KUKA KRL program: EPS_2_251806_MH42A_A_20260212042235.src

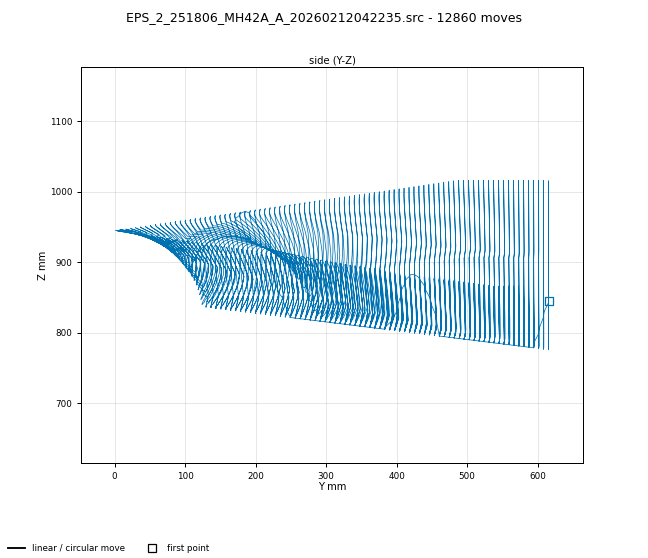
[picture p0: tool path of EPS_2_251806_MH42A_A_20260212042235.src, 12860 of 12862 moves have a stored position in this frame; points joined in program order, loops and branches not executed]
&ACCESS RVP
&REL 4
&COMMENT QRS 19112012
&PARAM EDITMASK = *
DEF PART()
EXT BAS (BAS_COMMAND :IN,REAL :IN )
INT I
BAS (#INITMOV,0 )

;KUKA QRS Post kuka4.cps  Date:22-06-2017 !

File_ID=3014

QRS_PRE_INIT()

;Init var - Until changes are made in qrs_pre_init
Outlet_Square_prg=0
Inlet_1_Square_prg=0
Inlet_2_Square_prg=0
Inlet_3_Square_prg=0
Inlet_4_Square_prg=0
Inlet_5_Square_prg=0

Outlet_1={X 0.000, Y 487.620, Z 915.500, B 0.000, E1 0.000 }
Inlet_1={X 0.000, Y 518.170, Z 495.500, B 0.000, E1 90.000 }
Inlet_2={X 0.000, Y 534.120, Z 275.500, B 0.000, E1 180.000 }
Outlet_1_type=201
Inlet_1_type=201
Inlet_2_type=201
;QRS#1=Sidecore dimensions
;QRS#2=200-8" PVC SDR 35
;QRS#3=200-8" PVC SDR 35
;QRS#4=200-8" PVC SDR 35
;QRS#5=
;QRS#6=
;QRS#7=
;QRS#8=
;QRS#9=12-08 PSX
;QRS#10=12-08 PSX
;QRS#11=12-08 PSX
;QRS#12=
;QRS#13=
;QRS#14=
;QRS#15=
;QRS#16=1220x127x1295 4,25'
;QRS#17=EPS Height
;QRS#18=1016
;QRS#19=*
;QRS#20= UPDATED VERSION 22-06-2017
;QRS#21=*
Outlet_Square=0100
Inlet_1_Square=0100
Inlet_2_Square=0100
Inlet_3_Square=0
Inlet_4_Square=0
Inlet_5_Square=0
Mill_Square=1
Outlet_Square_Prg=204
Inlet_1_Square_prg=204
Inlet_2_Square_prg=204

QRS_INIT()

$ADVANCE=5

; T1
PTP {E1 173.421,E2 173.421}
PTP {X 0,Y 615.492,A -85,B 0,C 180,E1 173.421,E2 173.421,E3 0,E4 0,E5 0,E6 0}
QRS_SPEED_INIT()
LIN {X 0,Y 615.492,Z 844.236,A -85,B 0,C 180,E1 173.421,E2 173.421,E3 0,E4 0,E5 0,E6 0} C_VEL
LIN {X 0,Y 615.497,Z 836.536,A -85,B 0,C 180,E1 172.455,E2 172.455} C_VEL
LIN {X 0,Y 615.498,Z 826.758,A -85,B 0,C 180,E1 171.463,E2 171.463} C_VEL
LIN {X 0,Y 615.497,Z 816.492,A -85,B 0,C 180,E1 170.636,E2 170.636} C_VEL
LIN {X 0,Y 615.425,Z 804.939,A -85,B 0,C 180,E1 169.888,E2 169.888} C_VEL
LIN {X 0,Y 615.422,Z 793.42,A -85,B 0,C 180,E1 169.306,E2 169.306} C_VEL
LIN {X 0,Y 615.465,Z 781.457,A -85,B 0,C 180,E1 168.848,E2 168.848} C_VEL
LIN {X 0,Y 615.493,Z 775.695,A -85,B 0,C 180,E1 168.661,E2 168.661} C_VEL
LIN {X 0,Y 615.444,Z 775.7,A -85,B 0,C 180,E1 166.085,E2 166.085} C_VEL
LIN {X 0,Y 615.403,Z 775.7,A -85,B 0,C 180,E1 163.411,E2 163.411} C_VEL
LIN {X 0,Y 615.452,Z 775.7,A -85,B 0,C 180,E1 160.661,E2 160.661} C_VEL
LIN {X 0,Y 615.44,Z 775.698,A -85,B 0,C 180,E1 157.862,E2 157.862} C_VEL
LIN {X 0,Y 615.435,Z 775.697,A -85,B 0,C 180,E1 155.726,E2 155.726} C_VEL
LIN {X 0,Y 615.428,Z 775.696,A -85,B 0,C 180,E1 153.553,E2 153.553} C_VEL
LIN {X 0,Y 615.422,Z 775.696,A -85,B 0,C 180,E1 151.338,E2 151.338} C_VEL
LIN {X 0,Y 615.421,Z 775.696,A -85,B 0,C 180,E1 149.076,E2 149.076} C_VEL
LIN {X 0,Y 615.455,Z 775.698,A -85,B 0,C 180,E1 146.471,E2 146.471} C_VEL
LIN {X 0,Y 615.47,Z 775.69,A -85,B 0,C 180,E1 143.574,E2 143.574} C_VEL
LIN {X 0,Y 615.434,Z 775.693,A -85,B 0,C 180,E1 140.945,E2 140.945} C_VEL
LIN {X 0,Y 615.446,Z 775.696,A -85,B 0,C 180,E1 138.522,E2 138.522} C_VEL
LIN {X 0,Y 615.495,Z 775.696,A -85,B 0,C 180,E1 135.851,E2 135.851} C_VEL
LIN {X 0,Y 615.457,Z 775.688,A -85,B 0,C 180,E1 133.044,E2 133.044} C_VEL
LIN {X 0,Y 615.447,Z 775.692,A -85,B 0,C 180,E1 130.61,E2 130.61} C_VEL
LIN {X 0,Y 615.476,Z 775.699,A -85,B 0,C 180,E1 128.01,E2 128.01} C_VEL
LIN {X 0,Y 615.492,Z 775.695,A -85,B 0,C 180,E1 125.616,E2 125.616} C_VEL
LIN {X 0,Y 615.487,Z 775.686,A -85,B 0,C 180,E1 123.237,E2 123.237} C_VEL
LIN {X 0,Y 615.481,Z 775.683,A -85,B 0,C 180,E1 120.921,E2 120.921} C_VEL
LIN {X 0,Y 615.463,Z 775.688,A -85,B 0,C 180,E1 118.445,E2 118.445} C_VEL
LIN {X 0,Y 615.492,Z 775.699,A -85,B 0,C 180,E1 115.716,E2 115.716} C_VEL
LIN {X 0,Y 615.492,Z 775.681,A -85,B 0,C 180,E1 112.845,E2 112.845} C_VEL
LIN {X 0,Y 615.467,Z 775.692,A -85,B 0,C 180,E1 110.034,E2 110.034} C_VEL
LIN {X 0,Y 615.484,Z 775.695,A -85,B 0,C 180,E1 107.272,E2 107.272} C_VEL
LIN {X 0,Y 615.492,Z 775.68,A -85,B 0,C 180,E1 104.55,E2 104.55} C_VEL
LIN {X 0,Y 615.474,Z 775.691,A -85,B 0,C 180,E1 101.862,E2 101.862} C_VEL
LIN {X 0,Y 615.485,Z 775.703,A -85,B 0,C 180,E1 101.236,E2 101.236} C_VEL
LIN {X 0,Y 615.474,Z 787.797,A -85,B 0,C 180,E1 100.836,E2 100.836} C_VEL
LIN {X 0,Y 615.486,Z 800.177,A -85,B 0,C 180,E1 100.279,E2 100.279} C_VEL
LIN {X 0,Y 615.484,Z 811.562,A -85,B 0,C 180,E1 99.614,E2 99.614} C_VEL
LIN {X 0,Y 615.498,Z 821.809,A -85,B 0,C 180,E1 98.868,E2 98.868} C_VEL
LIN {X 0,Y 615.498,Z 830.91,A -85,B 0,C 180,E1 98.042,E2 98.042} C_VEL
LIN {X 0,Y 615.497,Z 838.588,A -85,B 0,C 180,E1 97.217,E2 97.217} C_VEL
LIN {X 0,Y 615.497,Z 846.003,A -85,B 0,C 180,E1 96.228,E2 96.228} C_VEL
LIN {X 0,Y 615.497,Z 851.952,A -85,B 0,C 180,E1 95.242,E2 95.242} C_VEL
LIN {X 0,Y 615.493,Z 856.653,A -85,B 0,C 180,E1 94.258,E2 94.258} C_VEL
LIN {X 0,Y 615.494,Z 860.251,A -85,B 0,C 180,E1 93.274,E2 93.274} C_VEL
LIN {X 0,Y 615.496,Z 862.112,A -85,B 0,C 180,E1 92.619,E2 92.619} C_VEL
LIN {X 0,Y 615.497,Z 863.532,A -85,B 0,C 180,E1 91.964,E2 91.964} C_VEL
LIN {X 0,Y 615.496,Z 865.141,A -85,B 0,C 180,E1 90.655,E2 90.655} C_VEL
LIN {X 0,Y 615.495,Z 865.384,A -85,B 0,C 180,E1 90.001,E2 90.001} C_VEL
LIN {X 0,Y 615.495,Z 865.206,A -85,B 0,C 180,E1 89.347,E2 89.347} C_VEL
LIN {X 0,Y 615.497,Z 863.685,A -85,B 0,C 180,E1 88.038,E2 88.038} C_VEL
LIN {X 0,Y 615.498,Z 862.344,A -85,B 0,C 180,E1 87.383,E2 87.383} C_VEL
LIN {X 0,Y 615.496,Z 859.498,A -85,B 0,C 180,E1 86.401,E2 86.401} C_VEL
LIN {X 0,Y 615.499,Z 855.64,A -85,B 0,C 180,E1 85.417,E2 85.417} C_VEL
LIN {X 0,Y 615.498,Z 850.658,A -85,B 0,C 180,E1 84.432,E2 84.432} C_VEL
LIN {X 0,Y 615.489,Z 844.254,A -85,B 0,C 180,E1 83.424,E2 83.424} C_VEL
LIN {X 0,Y 615.497,Z 836.548,A -85,B 0,C 180,E1 82.456,E2 82.456} C_VEL
LIN {X 0,Y 615.498,Z 826.773,A -85,B 0,C 180,E1 81.465,E2 81.465} C_VEL
LIN {X 0,Y 615.498,Z 816.511,A -85,B 0,C 180,E1 80.637,E2 80.637} C_VEL
LIN {X 0,Y 615.486,Z 804.953,A -85,B 0,C 180,E1 79.89,E2 79.89} C_VEL
LIN {X 0,Y 615.473,Z 793.219,A -85,B 0,C 180,E1 79.299,E2 79.299} C_VEL
LIN {X 0,Y 615.472,Z 781.426,A -85,B 0,C 180,E1 78.847,E2 78.847} C_VEL
LIN {X 0,Y 615.483,Z 775.697,A -85,B 0,C 180,E1 78.662,E2 78.662} C_VEL
LIN {X 0,Y 615.482,Z 775.692,A -85,B 0,C 180,E1 76.071,E2 76.071} C_VEL
LIN {X 0,Y 615.486,Z 775.681,A -85,B 0,C 180,E1 73.415,E2 73.415} C_VEL
LIN {X 0,Y 615.474,Z 775.692,A -85,B 0,C 180,E1 70.663,E2 70.663} C_VEL
LIN {X 0,Y 615.478,Z 775.692,A -85,B 0,C 180,E1 67.865,E2 67.865} C_VEL
LIN {X 0,Y 615.487,Z 775.681,A -85,B 0,C 180,E1 65.01,E2 65.01} C_VEL
LIN {X 0,Y 615.484,Z 775.703,A -85,B 0,C 180,E1 62.087,E2 62.087} C_VEL
LIN {X 0,Y 615.486,Z 775.696,A -85,B 0,C 180,E1 59.842,E2 59.842} C_VEL
LIN {X 0,Y 615.475,Z 775.691,A -85,B 0,C 180,E1 57.544,E2 57.544} C_VEL
LIN {X 0,Y 615.474,Z 775.686,A -85,B 0,C 180,E1 55.186,E2 55.186} C_VEL
LIN {X 0,Y 615.49,Z 775.68,A -85,B 0,C 180,E1 52.76,E2 52.76} C_VEL
LIN {X 0,Y 615.489,Z 775.697,A -85,B 0,C 180,E1 49.911,E2 49.911} C_VEL
LIN {X 0,Y 615.494,Z 775.699,A -85,B 0,C 180,E1 47.65,E2 47.65} C_VEL
LIN {X 0,Y 615.47,Z 775.687,A -85,B 0,C 180,E1 44.932,E2 44.932} C_VEL
LIN {X 0,Y 615.484,Z 775.687,A -85,B 0,C 180,E1 42.082,E2 42.082} C_VEL
LIN {X 0,Y 615.487,Z 775.694,A -85,B 0,C 180,E1 39.75,E2 39.75} C_VEL
LIN {X 0,Y 615.465,Z 775.691,A -85,B 0,C 180,E1 36.937,E2 36.937} C_VEL
LIN {X 0,Y 615.463,Z 775.688,A -85,B 0,C 180,E1 34.701,E2 34.701} C_VEL
LIN {X 0,Y 615.475,Z 775.683,A -85,B 0,C 180,E1 32.332,E2 32.332} C_VEL
LIN {X 0,Y 615.486,Z 775.697,A -85,B 0,C 180,E1 29.407,E2 29.407} C_VEL
LIN {X 0,Y 615.484,Z 775.698,A -85,B 0,C 180,E1 27.049,E2 27.049} C_VEL
LIN {X 0,Y 615.461,Z 775.687,A -85,B 0,C 180,E1 24.273,E2 24.273} C_VEL
LIN {X 0,Y 615.486,Z 775.69,A -85,B 0,C 180,E1 21.432,E2 21.432} C_VEL
LIN {X 0,Y 615.463,Z 775.695,A -85,B 0,C 180,E1 18.604,E2 18.604} C_VEL
LIN {X 0,Y 615.462,Z 775.687,A -85,B 0,C 180,E1 15.906,E2 15.906} C_VEL
LIN {X 0,Y 615.492,Z 775.689,A -85,B 0,C 180,E1 13.201,E2 13.201} C_VEL
LIN {X 0,Y 615.47,Z 775.697,A -85,B 0,C 180,E1 10.527,E2 10.527} C_VEL
LIN {X 0,Y 615.476,Z 775.698,A -85,B 0,C 180,E1 8.537,E2 8.537} C_VEL
LIN {X 0,Y 615.447,Z 775.691,A -85,B 0,C 180,E1 5.899,E2 5.899} C_VEL
LIN {X 0,Y 615.479,Z 775.685,A -85,B 0,C 180,E1 3.273,E2 3.273} C_VEL
LIN {X 0,Y 615.491,Z 775.697,A -85,B 0,C 180,E1 0.654,E2 0.654} C_VEL
LIN {X 0,Y 615.453,Z 775.696,A -85,B 0,C 180,E1 -1.963,E2 -1.963} C_VEL
LIN {X 0,Y 615.458,Z 775.697,A -85,B 0,C 180,E1 -3.929,E2 -3.929} C_VEL
LIN {X 0,Y 615.465,Z 775.698,A -85,B 0,C 180,E1 -5.899,E2 -5.899} C_VEL
LIN {X 0,Y 615.438,Z 775.693,A -85,B 0,C 180,E1 -8.537,E2 -8.537} C_VEL
LIN {X 0,Y 615.475,Z 775.688,A -85,B 0,C 180,E1 -11.193,E2 -11.193} C_VEL
LIN {X 0,Y 615.483,Z 775.699,A -85,B 0,C 180,E1 -13.939,E2 -13.939} C_VEL
LIN {X 0,Y 615.432,Z 775.695,A -85,B 0,C 180,E1 -16.588,E2 -16.588} C_VEL
LIN {X 0,Y 615.432,Z 775.695,A -85,B 0,C 180,E1 -18.648,E2 -18.648} C_VEL
LIN {X 0,Y 615.43,Z 775.695,A -85,B 0,C 180,E1 -20.733,E2 -20.733} C_VEL
LIN {X 0,Y 615.428,Z 775.695,A -85,B 0,C 180,E1 -22.847,E2 -22.847} C_VEL
LIN {X 0,Y 615.424,Z 775.695,A -85,B 0,C 180,E1 -24.995,E2 -24.995} C_VEL
LIN {X 0,Y 615.427,Z 775.695,A -85,B 0,C 180,E1 -27.18,E2 -27.18} C_VEL
LIN {X 0,Y 615.47,Z 775.692,A -85,B 0,C 180,E1 -29.796,E2 -29.796} C_VEL
LIN {X 0,Y 615.47,Z 775.7,A -85,B 0,C 180,E1 -32.459,E2 -32.459} C_VEL
LIN {X 0,Y 615.437,Z 775.698,A -85,B 0,C 180,E1 -34.818,E2 -34.818} C_VEL
LIN {X 0,Y 615.417,Z 775.697,A -85,B 0,C 180,E1 -37.247,E2 -37.247} C_VEL
LIN {X 0,Y 615.461,Z 775.695,A -85,B 0,C 180,E1 -40.089,E2 -40.089} C_VEL
LIN {X 0,Y 615.431,Z 775.699,A -85,B 0,C 180,E1 -43.044,E2 -43.044} C_VEL
LIN {X 0,Y 615.433,Z 775.699,A -85,B 0,C 180,E1 -45.074,E2 -45.074} C_VEL
LIN {X 0,Y 615.451,Z 775.7,A -85,B 0,C 180,E1 -46.956,E2 -46.956} C_VEL
LIN {X 0,Y 615.415,Z 775.699,A -85,B 0,C 180,E1 -49.39,E2 -49.39} C_VEL
LIN {X 0,Y 615.408,Z 775.699,A -85,B 0,C 180,E1 -51.928,E2 -51.928} C_VEL
LIN {X 0,Y 615.43,Z 775.818,A -85,B 0,C 180,E1 -54.357,E2 -54.357} C_VEL
LIN {X 0,Y 615.479,Z 789.637,A -85,B 0,C 180,E1 -57.155,E2 -57.155} C_VEL
LIN {X 0,Y 615.478,Z 803.332,A -85,B 0,C 180,E1 -59.841,E2 -59.841} C_VEL
LIN {X 0,Y 615.456,Z 817.027,A -85,B 0,C 180,E1 -62.455,E2 -62.455} C_VEL
LIN {X 0,Y 615.491,Z 830.716,A -85,B 0,C 180,E1 -65.01,E2 -65.01} C_VEL
LIN {X 0,Y 615.47,Z 846.347,A -85,B 0,C 180,E1 -67.865,E2 -67.865} C_VEL
LIN {X 0,Y 615.451,Z 860.013,A -85,B 0,C 180,E1 -70.315,E2 -70.315} C_VEL
LIN {X 0,Y 615.481,Z 873.666,A -85,B 0,C 180,E1 -72.731,E2 -72.731} C_VEL
LIN {X 0,Y 615.489,Z 889.253,A -85,B 0,C 180,E1 -75.452,E2 -75.452} C_VEL
LIN {X 0,Y 615.464,Z 905.807,A -85,B 0,C 180,E1 -78.307,E2 -78.307} C_VEL
LIN {X 0,Y 615.477,Z 921.127,A -85,B 0,C 180,E1 -78.6,E2 -78.6} C_VEL
LIN {X 0,Y 615.49,Z 933.53,A -85,B 0,C 180,E1 -78.961,E2 -78.961} C_VEL
LIN {X 0,Y 615.489,Z 946.05,A -85,B 0,C 180,E1 -79.474,E2 -79.474} C_VEL
LIN {X 0,Y 615.485,Z 958.411,A -85,B 0,C 180,E1 -80.139,E2 -80.139} C_VEL
LIN {X 0,Y 615.498,Z 969.249,A -85,B 0,C 180,E1 -80.886,E2 -80.886} C_VEL
LIN {X 0,Y 615.499,Z 978.016,A -85,B 0,C 180,E1 -81.63,E2 -81.63} C_VEL
LIN {X 0,Y 615.498,Z 987.617,A -85,B 0,C 180,E1 -82.621,E2 -82.621} C_VEL
LIN {X 0,Y 615.491,Z 995.213,A -85,B 0,C 180,E1 -83.609,E2 -83.609} C_VEL
LIN {X 0,Y 615.498,Z 1002.211,A -85,B 0,C 180,E1 -84.76,E2 -84.76} C_VEL
LIN {X 0,Y 615.493,Z 1006.857,A -85,B 0,C 180,E1 -85.745,E2 -85.745} C_VEL
LIN {X 0,Y 615.494,Z 1010.403,A -85,B 0,C 180,E1 -86.728,E2 -86.728} C_VEL
LIN {X 0,Y 615.497,Z 1012.236,A -85,B 0,C 180,E1 -87.383,E2 -87.383} C_VEL
LIN {X 0,Y 615.497,Z 1013.61,A -85,B 0,C 180,E1 -88.038,E2 -88.038} C_VEL
LIN {X 0,Y 615.496,Z 1015.174,A -85,B 0,C 180,E1 -89.347,E2 -89.347} C_VEL
LIN {X 0,Y 615.494,Z 1015.389,A -85,B 0,C 180,E1 -90.001,E2 -90.001} C_VEL
LIN {X 0,Y 615.495,Z 1014.579,A -85,B 0,C 180,E1 -91.31,E2 -91.31} C_VEL
LIN {X 0,Y 615.497,Z 1013.606,A -85,B 0,C 180,E1 -91.964,E2 -91.964} C_VEL
LIN {X 0,Y 615.497,Z 1012.23,A -85,B 0,C 180,E1 -92.619,E2 -92.619} C_VEL
LIN {X 0,Y 615.496,Z 1009.346,A -85,B 0,C 180,E1 -93.602,E2 -93.602} C_VEL
LIN {X 0,Y 615.498,Z 1005.437,A -85,B 0,C 180,E1 -94.586,E2 -94.586} C_VEL
LIN {X 0,Y 615.499,Z 1000.399,A -85,B 0,C 180,E1 -95.571,E2 -95.571} C_VEL
LIN {X 0,Y 615.49,Z 993.913,A -85,B 0,C 180,E1 -96.578,E2 -96.578} C_VEL
LIN {X 0,Y 615.497,Z 986.123,A -85,B 0,C 180,E1 -97.546,E2 -97.546} C_VEL
LIN {X 0,Y 615.498,Z 976.245,A -85,B 0,C 180,E1 -98.538,E2 -98.538} C_VEL
LIN {X 0,Y 615.498,Z 965.851,A -85,B 0,C 180,E1 -99.365,E2 -99.365} C_VEL
LIN {X 0,Y 615.485,Z 955.558,A -85,B 0,C 180,E1 -100.029,E2 -100.029} C_VEL
LIN {X 0,Y 615.486,Z 944.115,A -85,B 0,C 180,E1 -100.617,E2 -100.617} C_VEL
LIN {X 0,Y 615.492,Z 932.321,A -85,B 0,C 180,E1 -101.078,E2 -101.078} C_VEL
LIN {X 0,Y 615.474,Z 919.198,A -85,B 0,C 180,E1 -101.445,E2 -101.445} C_VEL
LIN {X 0,Y 615.464,Z 905.793,A -85,B 0,C 180,E1 -101.695,E2 -101.695} C_VEL
LIN {X 0,Y 615.489,Z 889.239,A -85,B 0,C 180,E1 -104.55,E2 -104.55} C_VEL
LIN {X 0,Y 615.481,Z 873.652,A -85,B 0,C 180,E1 -107.272,E2 -107.272} C_VEL
LIN {X 0,Y 615.451,Z 859.999,A -85,B 0,C 180,E1 -109.687,E2 -109.687} C_VEL
LIN {X 0,Y 615.489,Z 845.179,A -85,B 0,C 180,E1 -112.346,E2 -112.346} C_VEL
LIN {X 0,Y 615.491,Z 830.702,A -85,B 0,C 180,E1 -114.992,E2 -114.992} C_VEL
LIN {X 0,Y 615.456,Z 817.013,A -85,B 0,C 180,E1 -117.548,E2 -117.548} C_VEL
LIN {X 0,Y 615.478,Z 803.318,A -85,B 0,C 180,E1 -120.161,E2 -120.161} C_VEL
LIN {X 0,Y 615.479,Z 789.623,A -85,B 0,C 180,E1 -122.847,E2 -122.847} C_VEL
LIN {X 0,Y 615.427,Z 775.7,A -85,B 0,C 180,E1 -125.671,E2 -125.671} C_VEL
LIN {X 0,Y 615.406,Z 775.7,A -85,B 0,C 180,E1 -128.075,E2 -128.075} C_VEL
LIN {X 0,Y 615.41,Z 775.7,A -85,B 0,C 180,E1 -130.613,E2 -130.613} C_VEL
LIN {X 0,Y 615.47,Z 775.7,A -85,B 0,C 180,E1 -133.247,E2 -133.247} C_VEL
LIN {X 0,Y 615.43,Z 775.699,A -85,B 0,C 180,E1 -136.009,E2 -136.009} C_VEL
LIN {X 0,Y 615.447,Z 775.699,A -85,B 0,C 180,E1 -137.925,E2 -137.925} C_VEL
LIN {X 0,Y 615.421,Z 775.699,A -85,B 0,C 180,E1 -140.245,E2 -140.245} C_VEL
LIN {X 0,Y 615.404,Z 775.699,A -85,B 0,C 180,E1 -142.752,E2 -142.752} C_VEL
LIN {X 0,Y 615.428,Z 775.7,A -85,B 0,C 180,E1 -145.308,E2 -145.308} C_VEL
LIN {X 0,Y 615.442,Z 775.698,A -85,B 0,C 180,E1 -148.312,E2 -148.312} C_VEL
LIN {X 0,Y 615.422,Z 775.699,A -85,B 0,C 180,E1 -150.59,E2 -150.59} C_VEL
LIN {X 0,Y 615.407,Z 775.699,A -85,B 0,C 180,E1 -152.971,E2 -152.971} C_VEL
LIN {X 0,Y 615.408,Z 775.699,A -85,B 0,C 180,E1 -155.005,E2 -155.005} C_VEL
LIN {X 0,Y 615.405,Z 775.699,A -85,B 0,C 180,E1 -157.152,E2 -157.152} C_VEL
LIN {X 0,Y 615.409,Z 775.699,A -85,B 0,C 180,E1 -159.464,E2 -159.464} C_VEL
LIN {X 0,Y 615.447,Z 775.701,A -85,B 0,C 180,E1 -162.042,E2 -162.042} C_VEL
LIN {X 0,Y 615.454,Z 775.698,A -85,B 0,C 180,E1 -164.773,E2 -164.773} C_VEL
LIN {X 0,Y 615.408,Z 775.698,A -85,B 0,C 180,E1 -167.468,E2 -167.468} C_VEL
LIN {X 0,Y 615.475,Z 775.741,A -85,B 0,C 180,E1 -168.765,E2 -168.765} C_VEL
LIN {X 0,Y 615.425,Z 788.344,A -85,B 0,C 180,E1 -169.184,E2 -169.184} C_VEL
LIN {X 0,Y 615.408,Z 800.209,A -85,B 0,C 180,E1 -169.721,E2 -169.721} C_VEL
LIN {X 0,Y 615.463,Z 811.581,A -85,B 0,C 180,E1 -170.386,E2 -170.386} C_VEL
LIN {X 0,Y 615.498,Z 821.823,A -85,B 0,C 180,E1 -171.133,E2 -171.133} C_VEL
LIN {X 0,Y 615.498,Z 830.921,A -85,B 0,C 180,E1 -171.959,E2 -171.959} C_VEL
LIN {X 0,Y 615.497,Z 838.597,A -85,B 0,C 180,E1 -172.784,E2 -172.784} C_VEL
LIN {X 0,Y 615.497,Z 846.011,A -85,B 0,C 180,E1 -173.773,E2 -173.773} C_VEL
LIN {X 0,Y 615.497,Z 851.958,A -85,B 0,C 180,E1 -174.759,E2 -174.759} C_VEL
LIN {X 0,Y 615.493,Z 856.658,A -85,B 0,C 180,E1 -175.744,E2 -175.744} C_VEL
LIN {X 0,Y 615.496,Z 860.254,A -85,B 0,C 180,E1 -176.727,E2 -176.727} C_VEL
LIN {X 0,Y 615.496,Z 862.115,A -85,B 0,C 180,E1 -177.382,E2 -177.382} C_VEL
LIN {X 0,Y 615.497,Z 863.534,A -85,B 0,C 180,E1 -178.037,E2 -178.037} C_VEL
LIN {X 0,Y 615.496,Z 865.142,A -85,B 0,C 180,E1 -179.346,E2 -179.346} C_VEL
LIN {X 0,Y 615.494,Z 865.384,A -85,B 0,C 180,E1 -180,E2 -180} C_VEL
LIN {X 0,Y 615.495,Z 865.206,A -85,B 0,C 180,E1 -180.654,E2 -180.654} C_VEL
LIN {X 0,Y 615.496,Z 863.683,A -85,B 0,C 180,E1 -181.963,E2 -181.963} C_VEL
LIN {X 0,Y 615.498,Z 862.341,A -85,B 0,C 180,E1 -182.618,E2 -182.618} C_VEL
LIN {X 0,Y 615.496,Z 859.494,A -85,B 0,C 180,E1 -183.601,E2 -183.601} C_VEL
LIN {X 0,Y 615.498,Z 855.634,A -85,B 0,C 180,E1 -184.585,E2 -184.585} C_VEL
LIN {X 0,Y 615.498,Z 850.651,A -85,B 0,C 180,E1 -185.57,E2 -185.57} C_VEL
LIN {X 0,Y 615.492,Z 844.236,A -85,B 0,C 180,E1 -186.579,E2 -186.579} C_VEL
LIN {X 0,Y 614.826,Z 841.054,A -85,B 0,C 180,E1 -187.028,E2 -187.028} C_VEL
LIN {X 0,Y 611.988,Z 835.48,A -85,B 0,C 180,E1 -187.745,E2 -187.745} C_VEL
LIN {X 0,Y 609.138,Z 829.207,A -85,B 0,C 180,E1 -188.426,E2 -188.426} C_VEL
LIN {X 0,Y 608.477,Z 824.966,A -85,B 0,C 180,E1 -188.816,E2 -188.816} C_VEL
LIN {X 0,Y 608.476,Z 814.391,A -85,B 0,C 180,E1 -189.641,E2 -189.641} C_VEL
LIN {X 0,Y 608.422,Z 803.602,A -85,B 0,C 180,E1 -190.314,E2 -190.314} C_VEL
LIN {X 0,Y 608.444,Z 791.79,A -85,B 0,C 180,E1 -190.893,E2 -190.893} C_VEL
LIN {X 0,Y 608.523,Z 778.958,A -85,B 0,C 180,E1 -191.365,E2 -191.365} C_VEL
LIN {X 0,Y 608.472,Z 776.695,A -85,B 0,C 180,E1 -191.45,E2 -191.45} C_VEL
LIN {X 0,Y 608.419,Z 776.694,A -85,B 0,C 180,E1 -194.039,E2 -194.039} C_VEL
LIN {X 0,Y 608.375,Z 776.696,A -85,B 0,C 180,E1 -196.498,E2 -196.498} C_VEL
LIN {X 0,Y 608.392,Z 776.695,A -85,B 0,C 180,E1 -198.872,E2 -198.872} C_VEL
LIN {X 0,Y 608.439,Z 776.7,A -85,B 0,C 180,E1 -201.693,E2 -201.693} C_VEL
LIN {X 0,Y 608.404,Z 776.693,A -85,B 0,C 180,E1 -204.573,E2 -204.573} C_VEL
LIN {X 0,Y 608.387,Z 776.695,A -85,B 0,C 180,E1 -206.777,E2 -206.777} C_VEL
LIN {X 0,Y 608.481,Z 776.694,A -85,B 0,C 180,E1 -209.779,E2 -209.779} C_VEL
LIN {X 0,Y 608.431,Z 776.69,A -85,B 0,C 180,E1 -212.517,E2 -212.517} C_VEL
LIN {X 0,Y 608.4,Z 776.693,A -85,B 0,C 180,E1 -214.898,E2 -214.898} C_VEL
LIN {X 0,Y 608.431,Z 776.69,A -85,B 0,C 180,E1 -217.153,E2 -217.153} C_VEL
LIN {X 0,Y 608.421,Z 776.693,A -85,B 0,C 180,E1 -219.444,E2 -219.444} C_VEL
LIN {X 0,Y 608.468,Z 776.69,A -85,B 0,C 180,E1 -222.334,E2 -222.334} C_VEL
LIN {X 0,Y 608.431,Z 776.69,A -85,B 0,C 180,E1 -224.799,E2 -224.799} C_VEL
LIN {X 0,Y 608.424,Z 776.69,A -85,B 0,C 180,E1 -227.037,E2 -227.037} C_VEL
LIN {X 0,Y 608.427,Z 776.694,A -85,B 0,C 180,E1 -229.694,E2 -229.694} C_VEL
LIN {X 0,Y 608.465,Z 776.695,A -85,B 0,C 180,E1 -232.253,E2 -232.253} C_VEL
LIN {X 0,Y 608.435,Z 776.689,A -85,B 0,C 180,E1 -235.097,E2 -235.097} C_VEL
LIN {X 0,Y 608.451,Z 776.692,A -85,B 0,C 180,E1 -237.904,E2 -237.904} C_VEL
LIN {X 0,Y 608.473,Z 776.694,A -85,B 0,C 180,E1 -240.22,E2 -240.22} C_VEL
LIN {X 0,Y 608.442,Z 776.688,A -85,B 0,C 180,E1 -243.225,E2 -243.225} C_VEL
LIN {X 0,Y 608.44,Z 776.691,A -85,B 0,C 180,E1 -245.856,E2 -245.856} C_VEL
LIN {X 0,Y 608.465,Z 776.694,A -85,B 0,C 180,E1 -248.307,E2 -248.307} C_VEL
LIN {X 0,Y 608.477,Z 776.684,A -85,B 0,C 180,E1 -251.283,E2 -251.283} C_VEL
LIN {X 0,Y 608.454,Z 776.688,A -85,B 0,C 180,E1 -253.905,E2 -253.905} C_VEL
LIN {X 0,Y 608.459,Z 776.696,A -85,B 0,C 180,E1 -256.642,E2 -256.642} C_VEL
LIN {X 0,Y 608.472,Z 776.695,A -85,B 0,C 180,E1 -258.654,E2 -258.654} C_VEL
LIN {X 0,Y 608.512,Z 788.579,A -85,B 0,C 180,E1 -259.063,E2 -259.063} C_VEL
LIN {X 0,Y 608.498,Z 800.342,A -85,B 0,C 180,E1 -259.602,E2 -259.602} C_VEL
LIN {X 0,Y 608.494,Z 811.769,A -85,B 0,C 180,E1 -260.274,E2 -260.274} C_VEL
LIN {X 0,Y 608.474,Z 822.067,A -85,B 0,C 180,E1 -261.028,E2 -261.028} C_VEL
LIN {X 0,Y 608.464,Z 831.232,A -85,B 0,C 180,E1 -261.865,E2 -261.865} C_VEL
LIN {X 0,Y 608.462,Z 838.957,A -85,B 0,C 180,E1 -262.699,E2 -262.699} C_VEL
LIN {X 0,Y 608.449,Z 846.429,A -85,B 0,C 180,E1 -263.699,E2 -263.699} C_VEL
LIN {X 0,Y 608.462,Z 852.429,A -85,B 0,C 180,E1 -264.697,E2 -264.697} C_VEL
LIN {X 0,Y 608.439,Z 857.174,A -85,B 0,C 180,E1 -265.693,E2 -265.693} C_VEL
LIN {X 0,Y 608.425,Z 860.809,A -85,B 0,C 180,E1 -266.688,E2 -266.688} C_VEL
LIN {X 0,Y 608.425,Z 862.687,A -85,B 0,C 180,E1 -267.351,E2 -267.351} C_VEL
LIN {X 0,Y 608.442,Z 864.125,A -85,B 0,C 180,E1 -268.013,E2 -268.013} C_VEL
LIN {X 0,Y 608.439,Z 865.751,A -85,B 0,C 180,E1 -269.337,E2 -269.337} C_VEL
LIN {X 0,Y 608.435,Z 865.995,A -85,B 0,C 180,E1 -269.999,E2 -269.999} C_VEL
LIN {X 0,Y 608.438,Z 865.816,A -85,B 0,C 180,E1 -270.661,E2 -270.661} C_VEL
LIN {X 0,Y 608.443,Z 864.278,A -85,B 0,C 180,E1 -271.985,E2 -271.985} C_VEL
LIN {X 0,Y 608.426,Z 862.921,A -85,B 0,C 180,E1 -272.647,E2 -272.647} C_VEL
LIN {X 0,Y 608.449,Z 860.046,A -85,B 0,C 180,E1 -273.641,E2 -273.641} C_VEL
LIN {X 0,Y 608.433,Z 856.148,A -85,B 0,C 180,E1 -274.637,E2 -274.637} C_VEL
LIN {X 0,Y 608.449,Z 851.12,A -85,B 0,C 180,E1 -275.633,E2 -275.633} C_VEL
LIN {X 0,Y 608.438,Z 844.804,A -85,B 0,C 180,E1 -276.632,E2 -276.632} C_VEL
LIN {X 0,Y 608.475,Z 836.888,A -85,B 0,C 180,E1 -277.632,E2 -277.632} C_VEL
LIN {X 0,Y 608.472,Z 827.043,A -85,B 0,C 180,E1 -278.634,E2 -278.634} C_VEL
LIN {X 0,Y 608.48,Z 816.734,A -85,B 0,C 180,E1 -279.472,E2 -279.472} C_VEL
LIN {X 0,Y 608.483,Z 805.124,A -85,B 0,C 180,E1 -280.228,E2 -280.228} C_VEL
LIN {X 0,Y 608.497,Z 793.336,A -85,B 0,C 180,E1 -280.825,E2 -280.825} C_VEL
LIN {X 0,Y 608.522,Z 781.413,A -85,B 0,C 180,E1 -281.285,E2 -281.285} C_VEL
LIN {X 0,Y 608.468,Z 776.696,A -85,B 0,C 180,E1 -281.449,E2 -281.449} C_VEL
LIN {X 0,Y 608.47,Z 776.688,A -85,B 0,C 180,E1 -284.036,E2 -284.036} C_VEL
LIN {X 0,Y 608.473,Z 776.684,A -85,B 0,C 180,E1 -286.782,E2 -286.782} C_VEL
LIN {X 0,Y 608.443,Z 776.696,A -85,B 0,C 180,E1 -289.569,E2 -289.569} C_VEL
LIN {X 0,Y 608.475,Z 776.685,A -85,B 0,C 180,E1 -292.404,E2 -292.404} C_VEL
LIN {X 0,Y 608.448,Z 776.688,A -85,B 0,C 180,E1 -294.57,E2 -294.57} C_VEL
LIN {X 0,Y 608.475,Z 776.685,A -85,B 0,C 180,E1 -297.206,E2 -297.206} C_VEL
LIN {X 0,Y 608.466,Z 776.697,A -85,B 0,C 180,E1 -299.971,E2 -299.971} C_VEL
LIN {X 0,Y 608.451,Z 776.69,A -85,B 0,C 180,E1 -302.52,E2 -302.52} C_VEL
LIN {X 0,Y 608.433,Z 776.689,A -85,B 0,C 180,E1 -305.276,E2 -305.276} C_VEL
LIN {X 0,Y 608.471,Z 776.688,A -85,B 0,C 180,E1 -307.744,E2 -307.744} C_VEL
LIN {X 0,Y 608.448,Z 776.697,A -85,B 0,C 180,E1 -310.328,E2 -310.328} C_VEL
LIN {X 0,Y 608.441,Z 776.689,A -85,B 0,C 180,E1 -312.958,E2 -312.958} C_VEL
LIN {X 0,Y 608.451,Z 776.688,A -85,B 0,C 180,E1 -315.734,E2 -315.734} C_VEL
LIN {X 0,Y 608.455,Z 776.694,A -85,B 0,C 180,E1 -318.656,E2 -318.656} C_VEL
LIN {X 0,Y 608.456,Z 776.686,A -85,B 0,C 180,E1 -321.411,E2 -321.411} C_VEL
LIN {X 0,Y 608.468,Z 776.686,A -85,B 0,C 180,E1 -323.949,E2 -323.949} C_VEL
LIN {X 0,Y 608.467,Z 776.69,A -85,B 0,C 180,E1 -326.329,E2 -326.329} C_VEL
LIN {X 0,Y 608.466,Z 776.696,A -85,B 0,C 180,E1 -328.726,E2 -328.726} C_VEL
LIN {X 0,Y 608.449,Z 776.689,A -85,B 0,C 180,E1 -331.38,E2 -331.38} C_VEL
LIN {X 0,Y 608.437,Z 776.688,A -85,B 0,C 180,E1 -333.964,E2 -333.964} C_VEL
LIN {X 0,Y 608.459,Z 776.686,A -85,B 0,C 180,E1 -336.155,E2 -336.155} C_VEL
LIN {X 0,Y 608.444,Z 776.698,A -85,B 0,C 180,E1 -339.018,E2 -339.018} C_VEL
LIN {X 0,Y 608.427,Z 776.69,A -85,B 0,C 180,E1 -341.827,E2 -341.827} C_VEL
LIN {X 0,Y 608.466,Z 776.688,A -85,B 0,C 180,E1 -344.594,E2 -344.594} C_VEL
LIN {X 0,Y 608.461,Z 776.694,A -85,B 0,C 180,E1 -347.323,E2 -347.323} C_VEL
LIN {X 0,Y 608.455,Z 776.695,A -85,B 0,C 180,E1 -349.35,E2 -349.35} C_VEL
LIN {X 0,Y 608.447,Z 776.688,A -85,B 0,C 180,E1 -352.033,E2 -352.033} C_VEL
LIN {X 0,Y 608.461,Z 776.687,A -85,B 0,C 180,E1 -354.698,E2 -354.698} C_VEL
LIN {X 0,Y 608.483,Z 776.693,A -85,B 0,C 180,E1 -357.352,E2 -357.352} C_VEL
LIN {X 0,Y 608.44,Z 776.691,A -85,B 0,C 180,E1 -360,E2 -360} C_VEL
LIN {X 0,Y 608.445,Z 776.688,A -85,B 0,C 180,E1 -362.648,E2 -362.648} C_VEL
LIN {X 0,Y 608.468,Z 776.69,A -85,B 0,C 180,E1 -365.302,E2 -365.302} C_VEL
LIN {X 0,Y 608.459,Z 776.692,A -85,B 0,C 180,E1 -367.967,E2 -367.967} C_VEL
LIN {X 0,Y 608.42,Z 776.691,A -85,B 0,C 180,E1 -370.651,E2 -370.651} C_VEL
LIN {X 0,Y 608.451,Z 776.69,A -85,B 0,C 180,E1 -373.357,E2 -373.357} C_VEL
LIN {X 0,Y 608.441,Z 776.695,A -85,B 0,C 180,E1 -376.094,E2 -376.094} C_VEL
LIN {X 0,Y 608.421,Z 776.69,A -85,B 0,C 180,E1 -378.871,E2 -378.871} C_VEL
LIN {X 0,Y 608.45,Z 776.692,A -85,B 0,C 180,E1 -381.692,E2 -381.692} C_VEL
LIN {X 0,Y 608.419,Z 776.694,A -85,B 0,C 180,E1 -384.573,E2 -384.573} C_VEL
LIN {X 0,Y 608.406,Z 776.692,A -85,B 0,C 180,E1 -387.198,E2 -387.198} C_VEL
LIN {X 0,Y 608.48,Z 776.69,A -85,B 0,C 180,E1 -389.977,E2 -389.977} C_VEL
LIN {X 0,Y 608.417,Z 776.693,A -85,B 0,C 180,E1 -392.882,E2 -392.882} C_VEL
LIN {X 0,Y 608.395,Z 776.694,A -85,B 0,C 180,E1 -395.281,E2 -395.281} C_VEL
LIN {X 0,Y 608.446,Z 776.695,A -85,B 0,C 180,E1 -398.241,E2 -398.241} C_VEL
LIN {X 0,Y 608.391,Z 776.695,A -85,B 0,C 180,E1 -401.182,E2 -401.182} C_VEL
LIN {X 0,Y 608.412,Z 776.692,A -85,B 0,C 180,E1 -403.306,E2 -403.306} C_VEL
LIN {X 0,Y 608.424,Z 776.693,A -85,B 0,C 180,E1 -406.129,E2 -406.129} C_VEL
LIN {X 0,Y 608.437,Z 776.698,A -85,B 0,C 180,E1 -408.824,E2 -408.824} C_VEL
LIN {X 0,Y 608.389,Z 776.696,A -85,B 0,C 180,E1 -411.408,E2 -411.408} C_VEL
LIN {X 0,Y 608.423,Z 776.698,A -85,B 0,C 180,E1 -413.085,E2 -413.085} C_VEL
LIN {X 0,Y 608.417,Z 776.817,A -85,B 0,C 180,E1 -414.091,E2 -414.091} C_VEL
LIN {X 0,Y 608.646,Z 781.454,A -85,B 0,C 180,E1 -415.068,E2 -415.068} C_VEL
LIN {X 0,Y 608.623,Z 794.35,A -85,B 0,C 180,E1 -417.686,E2 -417.686} C_VEL
LIN {X 0,Y 608.582,Z 807.245,A -85,B 0,C 180,E1 -420.228,E2 -420.228} C_VEL
LIN {X 0,Y 608.565,Z 821.69,A -85,B 0,C 180,E1 -423.004,E2 -423.004} C_VEL
LIN {X 0,Y 608.554,Z 835.972,A -85,B 0,C 180,E1 -425.684,E2 -425.684} C_VEL
LIN {X 0,Y 608.475,Z 850.285,A -85,B 0,C 180,E1 -428.31,E2 -428.31} C_VEL
LIN {X 0,Y 608.515,Z 866.713,A -85,B 0,C 180,E1 -431.273,E2 -431.273} C_VEL
LIN {X 0,Y 608.49,Z 881.587,A -85,B 0,C 180,E1 -433.908,E2 -433.908} C_VEL
LIN {X 0,Y 608.431,Z 897.238,A -85,B 0,C 180,E1 -436.644,E2 -436.644} C_VEL
LIN {X 0,Y 608.427,Z 906.189,A -85,B 0,C 180,E1 -438.191,E2 -438.191} C_VEL
LIN {X 0,Y 608.539,Z 919.413,A -85,B 0,C 180,E1 -438.426,E2 -438.426} C_VEL
LIN {X 0,Y 608.527,Z 932.253,A -85,B 0,C 180,E1 -438.787,E2 -438.787} C_VEL
LIN {X 0,Y 608.508,Z 944.298,A -85,B 0,C 180,E1 -439.261,E2 -439.261} C_VEL
LIN {X 0,Y 608.48,Z 955.778,A -85,B 0,C 180,E1 -439.856,E2 -439.856} C_VEL
LIN {X 0,Y 608.503,Z 967.27,A -85,B 0,C 180,E1 -440.612,E2 -440.612} C_VEL
LIN {X 0,Y 608.472,Z 976.551,A -85,B 0,C 180,E1 -441.366,E2 -441.366} C_VEL
LIN {X 0,Y 608.475,Z 986.489,A -85,B 0,C 180,E1 -442.368,E2 -442.368} C_VEL
LIN {X 0,Y 608.441,Z 994.716,A -85,B 0,C 180,E1 -443.401,E2 -443.401} C_VEL
LIN {X 0,Y 608.45,Z 1000.873,A -85,B 0,C 180,E1 -444.367,E2 -444.367} C_VEL
LIN {X 0,Y 608.432,Z 1005.955,A -85,B 0,C 180,E1 -445.363,E2 -445.363} C_VEL
LIN {X 0,Y 608.449,Z 1009.9,A -85,B 0,C 180,E1 -446.359,E2 -446.359} C_VEL
LIN {X 0,Y 608.425,Z 1012.812,A -85,B 0,C 180,E1 -447.353,E2 -447.353} C_VEL
LIN {X 0,Y 608.442,Z 1014.203,A -85,B 0,C 180,E1 -448.015,E2 -448.015} C_VEL
LIN {X 0,Y 608.438,Z 1015.784,A -85,B 0,C 180,E1 -449.339,E2 -449.339} C_VEL
LIN {X 0,Y 608.434,Z 1016,A -85,B 0,C 180,E1 -450.001,E2 -450.001} C_VEL
LIN {X 0,Y 608.448,Z 1015.182,A -85,B 0,C 180,E1 -451.325,E2 -451.325} C_VEL
LIN {X 0,Y 608.442,Z 1014.199,A -85,B 0,C 180,E1 -451.987,E2 -451.987} C_VEL
LIN {X 0,Y 608.425,Z 1012.806,A -85,B 0,C 180,E1 -452.649,E2 -452.649} C_VEL
LIN {X 0,Y 608.449,Z 1009.892,A -85,B 0,C 180,E1 -453.644,E2 -453.644} C_VEL
LIN {X 0,Y 608.432,Z 1005.945,A -85,B 0,C 180,E1 -454.639,E2 -454.639} C_VEL
LIN {X 0,Y 608.437,Z 999.87,A -85,B 0,C 180,E1 -455.802,E2 -455.802} C_VEL
LIN {X 0,Y 608.462,Z 993.227,A -85,B 0,C 180,E1 -456.8,E2 -456.8} C_VEL
LIN {X 0,Y 608.456,Z 984.979,A -85,B 0,C 180,E1 -457.801,E2 -457.801} C_VEL
LIN {X 0,Y 608.477,Z 974.586,A -85,B 0,C 180,E1 -458.804,E2 -458.804} C_VEL
LIN {X 0,Y 608.493,Z 963.731,A -85,B 0,C 180,E1 -459.642,E2 -459.642} C_VEL
LIN {X 0,Y 608.49,Z 952.753,A -85,B 0,C 180,E1 -460.314,E2 -460.314} C_VEL
LIN {X 0,Y 608.507,Z 940.876,A -85,B 0,C 180,E1 -460.886,E2 -460.886} C_VEL
LIN {X 0,Y 608.553,Z 928.848,A -85,B 0,C 180,E1 -461.323,E2 -461.323} C_VEL
LIN {X 0,Y 608.515,Z 916.457,A -85,B 0,C 180,E1 -461.641,E2 -461.641} C_VEL
LIN {X 0,Y 608.428,Z 906.151,A -85,B 0,C 180,E1 -461.811,E2 -461.811} C_VEL
LIN {X 0,Y 608.469,Z 889.399,A -85,B 0,C 180,E1 -464.722,E2 -464.722} C_VEL
LIN {X 0,Y 608.483,Z 873.748,A -85,B 0,C 180,E1 -467.477,E2 -467.477} C_VEL
LIN {X 0,Y 608.452,Z 860.053,A -85,B 0,C 180,E1 -469.923,E2 -469.923} C_VEL
LIN {X 0,Y 608.55,Z 844.404,A -85,B 0,C 180,E1 -472.761,E2 -472.761} C_VEL
LIN {X 0,Y 608.565,Z 828.349,A -85,B 0,C 180,E1 -475.739,E2 -475.739} C_VEL
LIN {X 0,Y 608.535,Z 815.056,A -85,B 0,C 180,E1 -478.263,E2 -478.263} C_VEL
LIN {X 0,Y 608.613,Z 801.401,A -85,B 0,C 180,E1 -480.915,E2 -480.915} C_VEL
LIN {X 0,Y 608.654,Z 789.623,A -85,B 0,C 180,E1 -483.263,E2 -483.263} C_VEL
LIN {X 0,Y 608.637,Z 778.029,A -85,B 0,C 180,E1 -485.642,E2 -485.642} C_VEL
LIN {X 0,Y 608.39,Z 776.698,A -85,B 0,C 180,E1 -485.976,E2 -485.976} C_VEL
LIN {X 0,Y 608.374,Z 776.696,A -85,B 0,C 180,E1 -488.229,E2 -488.229} C_VEL
LIN {X 0,Y 608.381,Z 776.695,A -85,B 0,C 180,E1 -490.321,E2 -490.321} C_VEL
LIN {X 0,Y 608.377,Z 776.696,A -85,B 0,C 180,E1 -492.325,E2 -492.325} C_VEL
LIN {X 0,Y 608.391,Z 776.694,A -85,B 0,C 180,E1 -494.257,E2 -494.257} C_VEL
LIN {X 0,Y 608.384,Z 776.695,A -85,B 0,C 180,E1 -496.701,E2 -496.701} C_VEL
LIN {X 0,Y 608.379,Z 776.696,A -85,B 0,C 180,E1 -498.817,E2 -498.817} C_VEL
LIN {X 0,Y 608.394,Z 776.7,A -85,B 0,C 180,E1 -501.406,E2 -501.406} C_VEL
LIN {X 0,Y 608.435,Z 776.696,A -85,B 0,C 180,E1 -503.957,E2 -503.957} C_VEL
LIN {X 0,Y 608.414,Z 776.694,A -85,B 0,C 180,E1 -506.326,E2 -506.326} C_VEL
LIN {X 0,Y 608.384,Z 776.695,A -85,B 0,C 180,E1 -508.743,E2 -508.743} C_VEL
LIN {X 0,Y 608.381,Z 776.695,A -85,B 0,C 180,E1 -510.975,E2 -510.975} C_VEL
LIN {X 0,Y 608.379,Z 776.696,A -85,B 0,C 180,E1 -513.222,E2 -513.222} C_VEL
LIN {X 0,Y 608.402,Z 776.694,A -85,B 0,C 180,E1 -515.427,E2 -515.427} C_VEL
LIN {X 0,Y 608.436,Z 776.699,A -85,B 0,C 180,E1 -518.307,E2 -518.307} C_VEL
LIN {X 0,Y 608.393,Z 776.694,A -85,B 0,C 180,E1 -521.128,E2 -521.128} C_VEL
LIN {X 0,Y 608.411,Z 776.695,A -85,B 0,C 180,E1 -523.905,E2 -523.905} C_VEL
LIN {X 0,Y 608.436,Z 776.697,A -85,B 0,C 180,E1 -526.643,E2 -526.643} C_VEL
LIN {X 0,Y 608.471,Z 776.694,A -85,B 0,C 180,E1 -528.655,E2 -528.655} C_VEL
LIN {X 0,Y 608.454,Z 788.367,A -85,B 0,C 180,E1 -529.054,E2 -529.054} C_VEL
LIN {X 0,Y 608.422,Z 800.36,A -85,B 0,C 180,E1 -529.602,E2 -529.602} C_VEL
LIN {X 0,Y 608.463,Z 811.785,A -85,B 0,C 180,E1 -530.275,E2 -530.275} C_VEL
LIN {X 0,Y 608.474,Z 822.082,A -85,B 0,C 180,E1 -531.029,E2 -531.029} C_VEL
LIN {X 0,Y 608.464,Z 831.242,A -85,B 0,C 180,E1 -531.866,E2 -531.866} C_VEL
LIN {X 0,Y 608.462,Z 838.964,A -85,B 0,C 180,E1 -532.701,E2 -532.701} C_VEL
LIN {X 0,Y 608.448,Z 846.435,A -85,B 0,C 180,E1 -533.7,E2 -533.7} C_VEL
LIN {X 0,Y 608.462,Z 852.433,A -85,B 0,C 180,E1 -534.698,E2 -534.698} C_VEL
LIN {X 0,Y 608.439,Z 857.177,A -85,B 0,C 180,E1 -535.694,E2 -535.694} C_VEL
LIN {X 0,Y 608.426,Z 860.811,A -85,B 0,C 180,E1 -536.689,E2 -536.689} C_VEL
LIN {X 0,Y 608.425,Z 862.691,A -85,B 0,C 180,E1 -537.352,E2 -537.352} C_VEL
LIN {X 0,Y 608.442,Z 864.127,A -85,B 0,C 180,E1 -538.014,E2 -538.014} C_VEL
LIN {X 0,Y 608.439,Z 865.752,A -85,B 0,C 180,E1 -539.338,E2 -539.338} C_VEL
LIN {X 0,Y 608.434,Z 865.995,A -85,B 0,C 180,E1 -540,E2 -540} C_VEL
LIN {X 0,Y 608.438,Z 865.815,A -85,B 0,C 180,E1 -540.662,E2 -540.662} C_VEL
LIN {X 0,Y 608.441,Z 864.276,A -85,B 0,C 180,E1 -541.986,E2 -541.986} C_VEL
LIN {X 0,Y 608.426,Z 862.917,A -85,B 0,C 180,E1 -542.648,E2 -542.648} C_VEL
LIN {X 0,Y 608.449,Z 860.04,A -85,B 0,C 180,E1 -543.642,E2 -543.642} C_VEL
LIN {X 0,Y 608.433,Z 856.141,A -85,B 0,C 180,E1 -544.638,E2 -544.638} C_VEL
LIN {X 0,Y 608.449,Z 851.111,A -85,B 0,C 180,E1 -545.634,E2 -545.634} C_VEL
LIN {X 0,Y 608.44,Z 844.794,A -85,B 0,C 180,E1 -546.633,E2 -546.633} C_VEL
LIN {X 0,Y 608.476,Z 836.878,A -85,B 0,C 180,E1 -547.633,E2 -547.633} C_VEL
LIN {X 0,Y 608.472,Z 827.03,A -85,B 0,C 180,E1 -548.636,E2 -548.636} C_VEL
LIN {X 0,Y 608.477,Z 824.966,A -85,B 0,C 180,E1 -548.816,E2 -548.816} C_VEL
LIN {X 0,Y 607.807,Z 820.632,A -85,B 0,C 180,E1 -549.187,E2 -549.187} C_VEL
LIN {X 0,Y 604.947,Z 813.391,A -85,B 0,C 180,E1 -549.766,E2 -549.766} C_VEL
LIN {X 0,Y 602.096,Z 805.768,A -85,B 0,C 180,E1 -550.299,E2 -550.299} C_VEL
LIN {X 0,Y 601.441,Z 800.697,A -85,B 0,C 180,E1 -550.592,E2 -550.592} C_VEL
LIN {X 0,Y 601.501,Z 788.677,A -85,B 0,C 180,E1 -551.153,E2 -551.153} C_VEL
LIN {X 0,Y 601.425,Z 777.578,A -85,B 0,C 180,E1 -551.544,E2 -551.544} C_VEL
LIN {X 0,Y 601.375,Z 777.57,A -85,B 0,C 180,E1 -554.207,E2 -554.207} C_VEL
LIN {X 0,Y 601.361,Z 777.572,A -85,B 0,C 180,E1 -556.988,E2 -556.988} C_VEL
LIN {X 0,Y 601.369,Z 777.577,A -85,B 0,C 180,E1 -559.811,E2 -559.811} C_VEL
LIN {X 0,Y 601.348,Z 777.572,A -85,B 0,C 180,E1 -562.589,E2 -562.589} C_VEL
LIN {X 0,Y 601.363,Z 777.57,A -85,B 0,C 180,E1 -564.88,E2 -564.88} C_VEL
LIN {X 0,Y 601.37,Z 777.573,A -85,B 0,C 180,E1 -567.353,E2 -567.353} C_VEL
LIN {X 0,Y 601.405,Z 777.569,A -85,B 0,C 180,E1 -570.165,E2 -570.165} C_VEL
LIN {X 0,Y 601.392,Z 777.566,A -85,B 0,C 180,E1 -572.71,E2 -572.71} C_VEL
LIN {X 0,Y 601.359,Z 777.571,A -85,B 0,C 180,E1 -575.106,E2 -575.106} C_VEL
LIN {X 0,Y 601.394,Z 777.569,A -85,B 0,C 180,E1 -577.422,E2 -577.422} C_VEL
LIN {X 0,Y 601.4,Z 777.576,A -85,B 0,C 180,E1 -579.996,E2 -579.996} C_VEL
LIN {X 0,Y 601.386,Z 777.568,A -85,B 0,C 180,E1 -582.673,E2 -582.673} C_VEL
LIN {X 0,Y 601.404,Z 777.567,A -85,B 0,C 180,E1 -585.479,E2 -585.479} C_VEL
LIN {X 0,Y 601.423,Z 777.568,A -85,B 0,C 180,E1 -588.407,E2 -588.407} C_VEL
LIN {X 0,Y 601.399,Z 777.566,A -85,B 0,C 180,E1 -590.872,E2 -590.872} C_VEL
LIN {X 0,Y 601.395,Z 777.566,A -85,B 0,C 180,E1 -593.416,E2 -593.416} C_VEL
LIN {X 0,Y 601.419,Z 777.571,A -85,B 0,C 180,E1 -596.067,E2 -596.067} C_VEL
LIN {X 0,Y 601.424,Z 777.568,A -85,B 0,C 180,E1 -598.545,E2 -598.545} C_VEL
LIN {X 0,Y 601.418,Z 777.563,A -85,B 0,C 180,E1 -601.372,E2 -601.372} C_VEL
LIN {X 0,Y 601.398,Z 777.566,A -85,B 0,C 180,E1 -603.635,E2 -603.635} C_VEL
LIN {X 0,Y 601.419,Z 777.57,A -85,B 0,C 180,E1 -606.589,E2 -606.589} C_VEL
LIN {X 0,Y 601.428,Z 777.562,A -85,B 0,C 180,E1 -609.477,E2 -609.477} C_VEL
LIN {X 0,Y 601.393,Z 777.575,A -85,B 0,C 180,E1 -612.311,E2 -612.311} C_VEL
LIN {X 0,Y 601.41,Z 777.574,A -85,B 0,C 180,E1 -614.408,E2 -614.408} C_VEL
LIN {X 0,Y 601.418,Z 777.565,A -85,B 0,C 180,E1 -617.171,E2 -617.171} C_VEL
LIN {X 0,Y 601.421,Z 777.574,A -85,B 0,C 180,E1 -618.541,E2 -618.541} C_VEL
LIN {X 0,Y 601.536,Z 789.758,A -85,B 0,C 180,E1 -618.984,E2 -618.984} C_VEL
LIN {X 0,Y 601.502,Z 800.337,A -85,B 0,C 180,E1 -619.48,E2 -619.48} C_VEL
LIN {X 0,Y 601.46,Z 811.771,A -85,B 0,C 180,E1 -620.159,E2 -620.159} C_VEL
LIN {X 0,Y 601.439,Z 822.069,A -85,B 0,C 180,E1 -620.923,E2 -620.923} C_VEL
LIN {X 0,Y 601.403,Z 831.249,A -85,B 0,C 180,E1 -621.769,E2 -621.769} C_VEL
LIN {X 0,Y 601.412,Z 838.964,A -85,B 0,C 180,E1 -622.613,E2 -622.613} C_VEL
LIN {X 0,Y 601.36,Z 846.338,A -85,B 0,C 180,E1 -623.61,E2 -623.61} C_VEL
LIN {X 0,Y 601.373,Z 852.434,A -85,B 0,C 180,E1 -624.634,E2 -624.634} C_VEL
LIN {X 0,Y 601.353,Z 857.177,A -85,B 0,C 180,E1 -625.642,E2 -625.642} C_VEL
LIN {X 0,Y 601.344,Z 860.811,A -85,B 0,C 180,E1 -626.649,E2 -626.649} C_VEL
LIN {X 0,Y 601.324,Z 862.689,A -85,B 0,C 180,E1 -627.319,E2 -627.319} C_VEL
LIN {X 0,Y 601.341,Z 864.122,A -85,B 0,C 180,E1 -627.99,E2 -627.99} C_VEL
LIN {X 0,Y 601.339,Z 865.752,A -85,B 0,C 180,E1 -629.329,E2 -629.329} C_VEL
LIN {X 0,Y 601.336,Z 865.989,A -85,B 0,C 180,E1 -629.999,E2 -629.999} C_VEL
LIN {X 0,Y 601.339,Z 865.816,A -85,B 0,C 180,E1 -630.668,E2 -630.668} C_VEL
LIN {X 0,Y 601.342,Z 864.277,A -85,B 0,C 180,E1 -632.008,E2 -632.008} C_VEL
LIN {X 0,Y 601.326,Z 862.92,A -85,B 0,C 180,E1 -632.678,E2 -632.678} C_VEL
LIN {X 0,Y 601.368,Z 860.045,A -85,B 0,C 180,E1 -633.684,E2 -633.684} C_VEL
LIN {X 0,Y 601.337,Z 856.148,A -85,B 0,C 180,E1 -634.691,E2 -634.691} C_VEL
LIN {X 0,Y 601.373,Z 851.119,A -85,B 0,C 180,E1 -635.7,E2 -635.7} C_VEL
LIN {X 0,Y 601.38,Z 844.799,A -85,B 0,C 180,E1 -636.71,E2 -636.71} C_VEL
LIN {X 0,Y 601.396,Z 836.878,A -85,B 0,C 180,E1 -637.722,E2 -637.722} C_VEL
LIN {X 0,Y 601.416,Z 827.024,A -85,B 0,C 180,E1 -638.737,E2 -638.737} C_VEL
LIN {X 0,Y 601.446,Z 816.73,A -85,B 0,C 180,E1 -639.584,E2 -639.584} C_VEL
LIN {X 0,Y 601.489,Z 805.12,A -85,B 0,C 180,E1 -640.348,E2 -640.348} C_VEL
LIN {X 0,Y 601.522,Z 794.174,A -85,B 0,C 180,E1 -640.915,E2 -640.915} C_VEL
LIN {X 0,Y 601.546,Z 782.436,A -85,B 0,C 180,E1 -641.383,E2 -641.383} C_VEL
LIN {X 0,Y 601.437,Z 777.572,A -85,B 0,C 180,E1 -641.563,E2 -641.563} C_VEL
LIN {X 0,Y 601.421,Z 777.565,A -85,B 0,C 180,E1 -644.204,E2 -644.204} C_VEL
LIN {X 0,Y 601.429,Z 777.563,A -85,B 0,C 180,E1 -646.984,E2 -646.984} C_VEL
LIN {X 0,Y 601.4,Z 777.575,A -85,B 0,C 180,E1 -649.808,E2 -649.808} C_VEL
LIN {X 0,Y 601.414,Z 777.564,A -85,B 0,C 180,E1 -652.604,E2 -652.604} C_VEL
LIN {X 0,Y 601.398,Z 777.565,A -85,B 0,C 180,E1 -654.877,E2 -654.877} C_VEL
LIN {X 0,Y 601.415,Z 777.574,A -85,B 0,C 180,E1 -657.866,E2 -657.866} C_VEL
LIN {X 0,Y 601.424,Z 777.57,A -85,B 0,C 180,E1 -660.162,E2 -660.162} C_VEL
LIN {X 0,Y 601.414,Z 777.565,A -85,B 0,C 180,E1 -662.714,E2 -662.714} C_VEL
LIN {X 0,Y 601.388,Z 777.567,A -85,B 0,C 180,E1 -665.11,E2 -665.11} C_VEL
LIN {X 0,Y 601.43,Z 777.562,A -85,B 0,C 180,E1 -667.417,E2 -667.417} C_VEL
LIN {X 0,Y 601.405,Z 777.571,A -85,B 0,C 180,E1 -669.993,E2 -669.993} C_VEL
LIN {X 0,Y 601.406,Z 777.569,A -85,B 0,C 180,E1 -672.668,E2 -672.668} C_VEL
LIN {X 0,Y 601.415,Z 777.563,A -85,B 0,C 180,E1 -675.481,E2 -675.481} C_VEL
LIN {X 0,Y 601.418,Z 777.574,A -85,B 0,C 180,E1 -678.405,E2 -678.405} C_VEL
LIN {X 0,Y 601.422,Z 777.567,A -85,B 0,C 180,E1 -680.874,E2 -680.874} C_VEL
LIN {X 0,Y 601.432,Z 777.561,A -85,B 0,C 180,E1 -683.732,E2 -683.732} C_VEL
LIN {X 0,Y 601.424,Z 777.573,A -85,B 0,C 180,E1 -686.686,E2 -686.686} C_VEL
LIN {X 0,Y 601.419,Z 777.568,A -85,B 0,C 180,E1 -689.058,E2 -689.058} C_VEL
LIN {X 0,Y 601.41,Z 777.566,A -85,B 0,C 180,E1 -691.372,E2 -691.372} C_VEL
LIN {X 0,Y 601.392,Z 777.566,A -85,B 0,C 180,E1 -693.636,E2 -693.636} C_VEL
LIN {X 0,Y 601.412,Z 777.569,A -85,B 0,C 180,E1 -696.589,E2 -696.589} C_VEL
LIN {X 0,Y 601.408,Z 777.567,A -85,B 0,C 180,E1 -699.477,E2 -699.477} C_VEL
LIN {X 0,Y 601.386,Z 777.568,A -85,B 0,C 180,E1 -702.311,E2 -702.311} C_VEL
LIN {X 0,Y 601.417,Z 777.574,A -85,B 0,C 180,E1 -705.103,E2 -705.103} C_VEL
LIN {X 0,Y 601.395,Z 777.567,A -85,B 0,C 180,E1 -707.857,E2 -707.857} C_VEL
LIN {X 0,Y 601.408,Z 777.565,A -85,B 0,C 180,E1 -709.904,E2 -709.904} C_VEL
LIN {X 0,Y 601.439,Z 777.561,A -85,B 0,C 180,E1 -712.615,E2 -712.615} C_VEL
LIN {X 0,Y 601.427,Z 777.573,A -85,B 0,C 180,E1 -715.308,E2 -715.308} C_VEL
LIN {X 0,Y 601.391,Z 777.568,A -85,B 0,C 180,E1 -717.991,E2 -717.991} C_VEL
LIN {X 0,Y 601.41,Z 777.567,A -85,B 0,C 180,E1 -720,E2 -720} C_VEL
LIN {X 0,Y 601.413,Z 777.564,A -85,B 0,C 180,E1 -722.679,E2 -722.679} C_VEL
LIN {X 0,Y 601.428,Z 777.568,A -85,B 0,C 180,E1 -725.364,E2 -725.364} C_VEL
LIN {X 0,Y 601.419,Z 777.567,A -85,B 0,C 180,E1 -728.061,E2 -728.061} C_VEL
LIN {X 0,Y 601.378,Z 777.568,A -85,B 0,C 180,E1 -730.777,E2 -730.777} C_VEL
LIN {X 0,Y 601.404,Z 777.57,A -85,B 0,C 180,E1 -733.516,E2 -733.516} C_VEL
LIN {X 0,Y 601.399,Z 777.569,A -85,B 0,C 180,E1 -736.288,E2 -736.288} C_VEL
LIN {X 0,Y 601.392,Z 777.566,A -85,B 0,C 180,E1 -739.1,E2 -739.1} C_VEL
LIN {X 0,Y 601.384,Z 777.578,A -85,B 0,C 180,E1 -741.96,E2 -741.96} C_VEL
LIN {X 0,Y 601.428,Z 777.569,A -85,B 0,C 180,E1 -744.295,E2 -744.295} C_VEL
LIN {X 0,Y 601.368,Z 777.569,A -85,B 0,C 180,E1 -747.115,E2 -747.115} C_VEL
LIN {X 0,Y 601.378,Z 777.568,A -85,B 0,C 180,E1 -749.395,E2 -749.395} C_VEL
LIN {X 0,Y 601.383,Z 777.57,A -85,B 0,C 180,E1 -751.728,E2 -751.728} C_VEL
LIN {X 0,Y 601.4,Z 777.573,A -85,B 0,C 180,E1 -754.12,E2 -754.12} C_VEL
LIN {X 0,Y 601.368,Z 777.577,A -85,B 0,C 180,E1 -756.586,E2 -756.586} C_VEL
LIN {X 0,Y 601.364,Z 777.571,A -85,B 0,C 180,E1 -759.13,E2 -759.13} C_VEL
LIN {X 0,Y 601.389,Z 777.567,A -85,B 0,C 180,E1 -761.768,E2 -761.768} C_VEL
LIN {X 0,Y 601.385,Z 777.578,A -85,B 0,C 180,E1 -764.534,E2 -764.534} C_VEL
LIN {X 0,Y 601.344,Z 777.574,A -85,B 0,C 180,E1 -767.326,E2 -767.326} C_VEL
LIN {X 0,Y 601.372,Z 777.57,A -85,B 0,C 180,E1 -769.432,E2 -769.432} C_VEL
LIN {X 0,Y 601.332,Z 777.575,A -85,B 0,C 180,E1 -771.728,E2 -771.728} C_VEL
LIN {X 0,Y 601.359,Z 777.675,A -85,B 0,C 180,E1 -773.807,E2 -773.807} C_VEL
LIN {X 0,Y 601.882,Z 781.409,A -85,B 0,C 180,E1 -774.608,E2 -774.608} C_VEL
LIN {X 0,Y 601.779,Z 794.15,A -85,B 0,C 180,E1 -777.232,E2 -777.232} C_VEL
LIN {X 0,Y 601.715,Z 807.245,A -85,B 0,C 180,E1 -779.854,E2 -779.854} C_VEL
LIN {X 0,Y 601.659,Z 821.297,A -85,B 0,C 180,E1 -782.593,E2 -782.593} C_VEL
LIN {X 0,Y 601.603,Z 834.634,A -85,B 0,C 180,E1 -785.132,E2 -785.132} C_VEL
LIN {X 0,Y 601.533,Z 848.428,A -85,B 0,C 180,E1 -787.704,E2 -787.704} C_VEL
LIN {X 0,Y 601.487,Z 862.023,A -85,B 0,C 180,E1 -790.195,E2 -790.195} C_VEL
LIN {X 0,Y 601.47,Z 875.718,A -85,B 0,C 180,E1 -792.666,E2 -792.666} C_VEL
LIN {X 0,Y 601.427,Z 891.369,A -85,B 0,C 180,E1 -795.451,E2 -795.451} C_VEL
LIN {X 0,Y 601.398,Z 906.189,A -85,B 0,C 180,E1 -798.051,E2 -798.051} C_VEL
LIN {X 0,Y 601.576,Z 918.498,A -85,B 0,C 180,E1 -798.268,E2 -798.268} C_VEL
LIN {X 0,Y 601.558,Z 931.301,A -85,B 0,C 180,E1 -798.624,E2 -798.624} C_VEL
LIN {X 0,Y 601.538,Z 943.853,A -85,B 0,C 180,E1 -799.115,E2 -799.115} C_VEL
LIN {X 0,Y 601.477,Z 955.779,A -85,B 0,C 180,E1 -799.737,E2 -799.737} C_VEL
LIN {X 0,Y 601.461,Z 967.271,A -85,B 0,C 180,E1 -800.501,E2 -800.501} C_VEL
LIN {X 0,Y 601.436,Z 976.552,A -85,B 0,C 180,E1 -801.264,E2 -801.264} C_VEL
LIN {X 0,Y 601.396,Z 986.489,A -85,B 0,C 180,E1 -802.278,E2 -802.278} C_VEL
LIN {X 0,Y 601.38,Z 994.48,A -85,B 0,C 180,E1 -803.29,E2 -803.29} C_VEL
LIN {X 0,Y 601.371,Z 1000.873,A -85,B 0,C 180,E1 -804.3,E2 -804.3} C_VEL
LIN {X 0,Y 601.336,Z 1005.955,A -85,B 0,C 180,E1 -805.309,E2 -805.309} C_VEL
LIN {X 0,Y 601.367,Z 1009.9,A -85,B 0,C 180,E1 -806.316,E2 -806.316} C_VEL
LIN {X 0,Y 601.325,Z 1012.812,A -85,B 0,C 180,E1 -807.322,E2 -807.322} C_VEL
LIN {X 0,Y 601.341,Z 1014.204,A -85,B 0,C 180,E1 -807.992,E2 -807.992} C_VEL
LIN {X 0,Y 601.339,Z 1015.784,A -85,B 0,C 180,E1 -809.332,E2 -809.332} C_VEL
LIN {X 0,Y 601.335,Z 1016,A -85,B 0,C 180,E1 -810.001,E2 -810.001} C_VEL
LIN {X 0,Y 601.347,Z 1015.183,A -85,B 0,C 180,E1 -811.341,E2 -811.341} C_VEL
LIN {X 0,Y 601.341,Z 1014.2,A -85,B 0,C 180,E1 -812.01,E2 -812.01} C_VEL
LIN {X 0,Y 601.325,Z 1012.806,A -85,B 0,C 180,E1 -812.681,E2 -812.681} C_VEL
LIN {X 0,Y 601.367,Z 1009.892,A -85,B 0,C 180,E1 -813.686,E2 -813.686} C_VEL
LIN {X 0,Y 601.336,Z 1005.945,A -85,B 0,C 180,E1 -814.694,E2 -814.694} C_VEL
LIN {X 0,Y 601.372,Z 999.87,A -85,B 0,C 180,E1 -815.87,E2 -815.87} C_VEL
LIN {X 0,Y 601.382,Z 993.227,A -85,B 0,C 180,E1 -816.881,E2 -816.881} C_VEL
LIN {X 0,Y 601.401,Z 984.98,A -85,B 0,C 180,E1 -817.893,E2 -817.893} C_VEL
LIN {X 0,Y 601.435,Z 974.586,A -85,B 0,C 180,E1 -818.908,E2 -818.908} C_VEL
LIN {X 0,Y 601.479,Z 963.732,A -85,B 0,C 180,E1 -819.755,E2 -819.755} C_VEL
LIN {X 0,Y 601.51,Z 952.754,A -85,B 0,C 180,E1 -820.435,E2 -820.435} C_VEL
LIN {X 0,Y 601.531,Z 940.887,A -85,B 0,C 180,E1 -821.013,E2 -821.013} C_VEL
LIN {X 0,Y 601.586,Z 928.848,A -85,B 0,C 180,E1 -821.456,E2 -821.456} C_VEL
LIN {X 0,Y 601.577,Z 916.457,A -85,B 0,C 180,E1 -821.777,E2 -821.777} C_VEL
LIN {X 0,Y 601.399,Z 906.151,A -85,B 0,C 180,E1 -821.951,E2 -821.951} C_VEL
LIN {X 0,Y 601.417,Z 889.399,A -85,B 0,C 180,E1 -824.898,E2 -824.898} C_VEL
LIN {X 0,Y 601.48,Z 873.748,A -85,B 0,C 180,E1 -827.687,E2 -827.687} C_VEL
LIN {X 0,Y 601.456,Z 860.053,A -85,B 0,C 180,E1 -830.165,E2 -830.165} C_VEL
LIN {X 0,Y 601.579,Z 844.402,A -85,B 0,C 180,E1 -833.04,E2 -833.04} C_VEL
LIN {X 0,Y 601.634,Z 829.122,A -85,B 0,C 180,E1 -835.91,E2 -835.91} C_VEL
LIN {X 0,Y 601.678,Z 815.056,A -85,B 0,C 180,E1 -838.615,E2 -838.615} C_VEL
LIN {X 0,Y 601.751,Z 801.86,A -85,B 0,C 180,E1 -841.215,E2 -841.215} C_VEL
LIN {X 0,Y 601.839,Z 789.874,A -85,B 0,C 180,E1 -843.638,E2 -843.638} C_VEL
LIN {X 0,Y 601.805,Z 779.841,A -85,B 0,C 180,E1 -845.727,E2 -845.727} C_VEL
LIN {X 0,Y 601.349,Z 777.578,A -85,B 0,C 180,E1 -846.253,E2 -846.253} C_VEL
LIN {X 0,Y 601.354,Z 777.572,A -85,B 0,C 180,E1 -848.461,E2 -848.461} C_VEL
LIN {X 0,Y 601.36,Z 777.574,A -85,B 0,C 180,E1 -850.88,E2 -850.88} C_VEL
LIN {X 0,Y 601.405,Z 777.573,A -85,B 0,C 180,E1 -853.589,E2 -853.589} C_VEL
LIN {X 0,Y 601.338,Z 777.573,A -85,B 0,C 180,E1 -856.437,E2 -856.437} C_VEL
LIN {X 0,Y 601.346,Z 777.575,A -85,B 0,C 180,E1 -859.12,E2 -859.12} C_VEL
LIN {X 0,Y 601.37,Z 777.58,A -85,B 0,C 180,E1 -861.728,E2 -861.728} C_VEL
LIN {X 0,Y 601.364,Z 777.573,A -85,B 0,C 180,E1 -864.244,E2 -864.244} C_VEL
LIN {X 0,Y 601.361,Z 777.57,A -85,B 0,C 180,E1 -866.682,E2 -866.682} C_VEL
LIN {X 0,Y 601.359,Z 777.57,A -85,B 0,C 180,E1 -869.054,E2 -869.054} C_VEL
LIN {X 0,Y 601.353,Z 777.573,A -85,B 0,C 180,E1 -871.369,E2 -871.369} C_VEL
LIN {X 0,Y 601.394,Z 777.572,A -85,B 0,C 180,E1 -874.381,E2 -874.381} C_VEL
LIN {X 0,Y 601.362,Z 777.574,A -85,B 0,C 180,E1 -876.587,E2 -876.587} C_VEL
LIN {X 0,Y 601.365,Z 777.57,A -85,B 0,C 180,E1 -879.476,E2 -879.476} C_VEL
LIN {X 0,Y 601.36,Z 777.581,A -85,B 0,C 180,E1 -882.311,E2 -882.311} C_VEL
LIN {X 0,Y 601.367,Z 777.571,A -85,B 0,C 180,E1 -885.101,E2 -885.101} C_VEL
LIN {X 0,Y 601.37,Z 777.57,A -85,B 0,C 180,E1 -887.857,E2 -887.857} C_VEL
LIN {X 0,Y 601.433,Z 777.573,A -85,B 0,C 180,E1 -888.542,E2 -888.542} C_VEL
LIN {X 0,Y 601.476,Z 790.483,A -85,B 0,C 180,E1 -889.014,E2 -889.014} C_VEL
LIN {X 0,Y 601.416,Z 801.927,A -85,B 0,C 180,E1 -889.564,E2 -889.564} C_VEL
LIN {X 0,Y 601.434,Z 813.066,A -85,B 0,C 180,E1 -890.245,E2 -890.245} C_VEL
LIN {X 0,Y 601.448,Z 823.116,A -85,B 0,C 180,E1 -891.008,E2 -891.008} C_VEL
LIN {X 0,Y 601.407,Z 832.957,A -85,B 0,C 180,E1 -891.939,E2 -891.939} C_VEL
LIN {X 0,Y 601.389,Z 840.327,A -85,B 0,C 180,E1 -892.783,E2 -892.783} C_VEL
LIN {X 0,Y 601.374,Z 847.501,A -85,B 0,C 180,E1 -893.787,E2 -893.787} C_VEL
LIN {X 0,Y 601.372,Z 852.433,A -85,B 0,C 180,E1 -894.635,E2 -894.635} C_VEL
LIN {X 0,Y 601.353,Z 857.174,A -85,B 0,C 180,E1 -895.643,E2 -895.643} C_VEL
LIN {X 0,Y 601.346,Z 860.809,A -85,B 0,C 180,E1 -896.65,E2 -896.65} C_VEL
LIN {X 0,Y 601.324,Z 862.694,A -85,B 0,C 180,E1 -897.32,E2 -897.32} C_VEL
LIN {X 0,Y 601.341,Z 864.128,A -85,B 0,C 180,E1 -897.991,E2 -897.991} C_VEL
LIN {X 0,Y 601.339,Z 865.753,A -85,B 0,C 180,E1 -899.33,E2 -899.33} C_VEL
LIN {X 0,Y 601.335,Z 865.996,A -85,B 0,C 180,E1 -900,E2 -900} C_VEL
LIN {X 0,Y 601.339,Z 865.815,A -85,B 0,C 180,E1 -900.67,E2 -900.67} C_VEL
LIN {X 0,Y 601.34,Z 864.276,A -85,B 0,C 180,E1 -902.009,E2 -902.009} C_VEL
LIN {X 0,Y 601.326,Z 862.909,A -85,B 0,C 180,E1 -902.68,E2 -902.68} C_VEL
LIN {X 0,Y 601.368,Z 860.033,A -85,B 0,C 180,E1 -903.685,E2 -903.685} C_VEL
LIN {X 0,Y 601.337,Z 856.134,A -85,B 0,C 180,E1 -904.693,E2 -904.693} C_VEL
LIN {X 0,Y 601.373,Z 851.105,A -85,B 0,C 180,E1 -905.701,E2 -905.701} C_VEL
LIN {X 0,Y 601.382,Z 844.79,A -85,B 0,C 180,E1 -906.711,E2 -906.711} C_VEL
LIN {X 0,Y 601.396,Z 836.873,A -85,B 0,C 180,E1 -907.723,E2 -907.723} C_VEL
LIN {X 0,Y 601.417,Z 827.013,A -85,B 0,C 180,E1 -908.738,E2 -908.738} C_VEL
LIN {X 0,Y 601.466,Z 816.708,A -85,B 0,C 180,E1 -909.585,E2 -909.585} C_VEL
LIN {X 0,Y 601.426,Z 805.095,A -85,B 0,C 180,E1 -910.35,E2 -910.35} C_VEL
LIN {X 0,Y 601.441,Z 800.697,A -85,B 0,C 180,E1 -910.592,E2 -910.592} C_VEL
LIN {X 0,Y 600.786,Z 797.296,A -85,B 0,C 180,E1 -910.782,E2 -910.782} C_VEL
LIN {X 0,Y 598.002,Z 791.997,A -85,B 0,C 180,E1 -911.084,E2 -911.084} C_VEL
LIN {X 0,Y 595.217,Z 786.547,A -85,B 0,C 180,E1 -911.357,E2 -911.357} C_VEL
LIN {X 0,Y 594.554,Z 782.914,A -85,B 0,C 180,E1 -911.501,E2 -911.501} C_VEL
LIN {X 0,Y 594.385,Z 778.449,A -85,B 0,C 180,E1 -911.661,E2 -911.661} C_VEL
LIN {X 0,Y 594.337,Z 778.446,A -85,B 0,C 180,E1 -914.378,E2 -914.378} C_VEL
LIN {X 0,Y 594.314,Z 778.452,A -85,B 0,C 180,E1 -917.196,E2 -917.196} C_VEL
LIN {X 0,Y 594.331,Z 778.449,A -85,B 0,C 180,E1 -920.055,E2 -920.055} C_VEL
LIN {X 0,Y 594.322,Z 778.448,A -85,B 0,C 180,E1 -922.969,E2 -922.969} C_VEL
LIN {X 0,Y 594.326,Z 778.449,A -85,B 0,C 180,E1 -925.195,E2 -925.195} C_VEL
LIN {X 0,Y 594.328,Z 778.452,A -85,B 0,C 180,E1 -927.515,E2 -927.515} C_VEL
LIN {X 0,Y 594.369,Z 778.444,A -85,B 0,C 180,E1 -930.324,E2 -930.324} C_VEL
LIN {X 0,Y 594.34,Z 778.444,A -85,B 0,C 180,E1 -932.953,E2 -932.953} C_VEL
LIN {X 0,Y 594.314,Z 778.451,A -85,B 0,C 180,E1 -935.412,E2 -935.412} C_VEL
LIN {X 0,Y 594.372,Z 778.452,A -85,B 0,C 180,E1 -937.942,E2 -937.942} C_VEL
LIN {X 0,Y 594.359,Z 778.443,A -85,B 0,C 180,E1 -940.819,E2 -940.819} C_VEL
LIN {X 0,Y 594.348,Z 778.445,A -85,B 0,C 180,E1 -943.302,E2 -943.302} C_VEL
LIN {X 0,Y 594.366,Z 778.451,A -85,B 0,C 180,E1 -946.161,E2 -946.161} C_VEL
LIN {X 0,Y 594.371,Z 778.441,A -85,B 0,C 180,E1 -949.179,E2 -949.179} C_VEL
LIN {X 0,Y 594.38,Z 778.449,A -85,B 0,C 180,E1 -952.058,E2 -952.058} C_VEL
LIN {X 0,Y 594.353,Z 778.446,A -85,B 0,C 180,E1 -954.677,E2 -954.677} C_VEL
LIN {X 0,Y 594.379,Z 778.44,A -85,B 0,C 180,E1 -957.089,E2 -957.089} C_VEL
LIN {X 0,Y 594.373,Z 778.442,A -85,B 0,C 180,E1 -959.675,E2 -959.675} C_VEL
LIN {X 0,Y 594.382,Z 778.446,A -85,B 0,C 180,E1 -962.539,E2 -962.539} C_VEL
LIN {X 0,Y 594.379,Z 778.443,A -85,B 0,C 180,E1 -964.806,E2 -964.806} C_VEL
LIN {X 0,Y 594.371,Z 778.441,A -85,B 0,C 180,E1 -967.264,E2 -967.264} C_VEL
LIN {X 0,Y 594.372,Z 778.444,A -85,B 0,C 180,E1 -969.945,E2 -969.945} C_VEL
LIN {X 0,Y 594.386,Z 778.445,A -85,B 0,C 180,E1 -972.806,E2 -972.806} C_VEL
LIN {X 0,Y 594.383,Z 778.441,A -85,B 0,C 180,E1 -975.83,E2 -975.83} C_VEL
LIN {X 0,Y 594.369,Z 778.45,A -85,B 0,C 180,E1 -978.424,E2 -978.424} C_VEL
LIN {X 0,Y 594.595,Z 782.611,A -85,B 0,C 180,E1 -978.58,E2 -978.58} C_VEL
LIN {X 0,Y 594.568,Z 793.871,A -85,B 0,C 180,E1 -979.033,E2 -979.033} C_VEL
LIN {X 0,Y 594.471,Z 806.422,A -85,B 0,C 180,E1 -979.698,E2 -979.698} C_VEL
LIN {X 0,Y 594.415,Z 817.784,A -85,B 0,C 180,E1 -980.471,E2 -980.471} C_VEL
LIN {X 0,Y 594.378,Z 827.84,A -85,B 0,C 180,E1 -981.328,E2 -981.328} C_VEL
LIN {X 0,Y 594.348,Z 837.552,A -85,B 0,C 180,E1 -982.354,E2 -982.354} C_VEL
LIN {X 0,Y 594.301,Z 845.423,A -85,B 0,C 180,E1 -983.393,E2 -983.393} C_VEL
LIN {X 0,Y 594.289,Z 852.439,A -85,B 0,C 180,E1 -984.57,E2 -984.57} C_VEL
LIN {X 0,Y 594.27,Z 857.181,A -85,B 0,C 180,E1 -985.59,E2 -985.59} C_VEL
LIN {X 0,Y 594.267,Z 860.814,A -85,B 0,C 180,E1 -986.609,E2 -986.609} C_VEL
LIN {X 0,Y 594.225,Z 862.69,A -85,B 0,C 180,E1 -987.287,E2 -987.287} C_VEL
LIN {X 0,Y 594.24,Z 864.114,A -85,B 0,C 180,E1 -987.966,E2 -987.966} C_VEL
LIN {X 0,Y 594.247,Z 865.131,A -85,B 0,C 180,E1 -988.643,E2 -988.643} C_VEL
LIN {X 0,Y 594.24,Z 865.752,A -85,B 0,C 180,E1 -989.321,E2 -989.321} C_VEL
LIN {X 0,Y 594.239,Z 865.816,A -85,B 0,C 180,E1 -990.676,E2 -990.676} C_VEL
LIN {X 0,Y 594.24,Z 864.277,A -85,B 0,C 180,E1 -992.032,E2 -992.032} C_VEL
LIN {X 0,Y 594.226,Z 862.919,A -85,B 0,C 180,E1 -992.71,E2 -992.71} C_VEL
LIN {X 0,Y 594.289,Z 860.044,A -85,B 0,C 180,E1 -993.728,E2 -993.728} C_VEL
LIN {X 0,Y 594.242,Z 856.147,A -85,B 0,C 180,E1 -994.748,E2 -994.748} C_VEL
LIN {X 0,Y 594.299,Z 851.118,A -85,B 0,C 180,E1 -995.768,E2 -995.768} C_VEL
LIN {X 0,Y 594.315,Z 844.794,A -85,B 0,C 180,E1 -996.79,E2 -996.79} C_VEL
LIN {X 0,Y 594.346,Z 836.869,A -85,B 0,C 180,E1 -997.814,E2 -997.814} C_VEL
LIN {X 0,Y 594.366,Z 828.787,A -85,B 0,C 180,E1 -998.67,E2 -998.67} C_VEL
LIN {X 0,Y 594.419,Z 820.034,A -85,B 0,C 180,E1 -999.441,E2 -999.441} C_VEL
LIN {X 0,Y 594.445,Z 810.586,A -85,B 0,C 180,E1 -1000.128,E2 -1000.128} C_VEL
LIN {X 0,Y 594.541,Z 800.445,A -85,B 0,C 180,E1 -1000.728,E2 -1000.728} C_VEL
LIN {X 0,Y 594.556,Z 788.497,A -85,B 0,C 180,E1 -1001.291,E2 -1001.291} C_VEL
LIN {X 0,Y 594.392,Z 778.448,A -85,B 0,C 180,E1 -1001.659,E2 -1001.659} C_VEL
LIN {X 0,Y 594.39,Z 778.439,A -85,B 0,C 180,E1 -1004.376,E2 -1004.376} C_VEL
LIN {X 0,Y 594.387,Z 778.442,A -85,B 0,C 180,E1 -1007.192,E2 -1007.192} C_VEL
LIN {X 0,Y 594.372,Z 778.446,A -85,B 0,C 180,E1 -1010.052,E2 -1010.052} C_VEL
LIN {X 0,Y 594.363,Z 778.442,A -85,B 0,C 180,E1 -1012.966,E2 -1012.966} C_VEL
LIN {X 0,Y 594.372,Z 778.442,A -85,B 0,C 180,E1 -1015.191,E2 -1015.191} C_VEL
LIN {X 0,Y 594.382,Z 778.444,A -85,B 0,C 180,E1 -1017.525,E2 -1017.525} C_VEL
LIN {X 0,Y 594.383,Z 778.444,A -85,B 0,C 180,E1 -1020.327,E2 -1020.327} C_VEL
LIN {X 0,Y 594.372,Z 778.441,A -85,B 0,C 180,E1 -1022.949,E2 -1022.949} C_VEL
LIN {X 0,Y 594.348,Z 778.445,A -85,B 0,C 180,E1 -1025.407,E2 -1025.407} C_VEL
LIN {X 0,Y 594.384,Z 778.446,A -85,B 0,C 180,E1 -1027.939,E2 -1027.939} C_VEL
LIN {X 0,Y 594.374,Z 778.443,A -85,B 0,C 180,E1 -1030.821,E2 -1030.821} C_VEL
LIN {X 0,Y 594.373,Z 778.444,A -85,B 0,C 180,E1 -1033.84,E2 -1033.84} C_VEL
LIN {X 0,Y 594.369,Z 778.446,A -85,B 0,C 180,E1 -1036.7,E2 -1036.7} C_VEL
LIN {X 0,Y 594.378,Z 778.44,A -85,B 0,C 180,E1 -1039.433,E2 -1039.433} C_VEL
LIN {X 0,Y 594.38,Z 778.448,A -85,B 0,C 180,E1 -1042.39,E2 -1042.39} C_VEL
LIN {X 0,Y 594.37,Z 778.451,A -85,B 0,C 180,E1 -1044.671,E2 -1044.671} C_VEL
LIN {X 0,Y 594.366,Z 778.445,A -85,B 0,C 180,E1 -1047.087,E2 -1047.087} C_VEL
LIN {X 0,Y 594.387,Z 778.438,A -85,B 0,C 180,E1 -1049.668,E2 -1049.668} C_VEL
LIN {X 0,Y 594.376,Z 778.447,A -85,B 0,C 180,E1 -1052.539,E2 -1052.539} C_VEL
LIN {X 0,Y 594.369,Z 778.451,A -85,B 0,C 180,E1 -1054.806,E2 -1054.806} C_VEL
LIN {X 0,Y 594.35,Z 778.448,A -85,B 0,C 180,E1 -1057.263,E2 -1057.263} C_VEL
LIN {X 0,Y 594.359,Z 778.442,A -85,B 0,C 180,E1 -1059.946,E2 -1059.946} C_VEL
LIN {X 0,Y 594.375,Z 778.447,A -85,B 0,C 180,E1 -1062.806,E2 -1062.806} C_VEL
LIN {X 0,Y 594.37,Z 778.442,A -85,B 0,C 180,E1 -1065.826,E2 -1065.826} C_VEL
LIN {X 0,Y 594.435,Z 778.438,A -85,B 0,C 180,E1 -1068.894,E2 -1068.894} C_VEL
LIN {X 0,Y 594.394,Z 778.44,A -85,B 0,C 180,E1 -1071.843,E2 -1071.843} C_VEL
LIN {X 0,Y 594.381,Z 778.44,A -85,B 0,C 180,E1 -1074.572,E2 -1074.572} C_VEL
LIN {X 0,Y 594.409,Z 778.445,A -85,B 0,C 180,E1 -1077.289,E2 -1077.289} C_VEL
LIN {X 0,Y 594.38,Z 778.442,A -85,B 0,C 180,E1 -1080,E2 -1080} C_VEL
LIN {X 0,Y 594.381,Z 778.44,A -85,B 0,C 180,E1 -1082.711,E2 -1082.711} C_VEL
LIN {X 0,Y 594.388,Z 778.447,A -85,B 0,C 180,E1 -1085.428,E2 -1085.428} C_VEL
LIN {X 0,Y 594.391,Z 778.441,A -85,B 0,C 180,E1 -1088.157,E2 -1088.157} C_VEL
LIN {X 0,Y 594.358,Z 778.443,A -85,B 0,C 180,E1 -1091.068,E2 -1091.068} C_VEL
LIN {X 0,Y 594.366,Z 778.45,A -85,B 0,C 180,E1 -1093.679,E2 -1093.679} C_VEL
LIN {X 0,Y 594.327,Z 778.447,A -85,B 0,C 180,E1 -1096.704,E2 -1096.704} C_VEL
LIN {X 0,Y 594.345,Z 778.446,A -85,B 0,C 180,E1 -1099.335,E2 -1099.335} C_VEL
LIN {X 0,Y 594.339,Z 778.448,A -85,B 0,C 180,E1 -1101.504,E2 -1101.504} C_VEL
LIN {X 0,Y 594.372,Z 778.445,A -85,B 0,C 180,E1 -1104.447,E2 -1104.447} C_VEL
LIN {X 0,Y 594.334,Z 778.447,A -85,B 0,C 180,E1 -1106.702,E2 -1106.702} C_VEL
LIN {X 0,Y 594.355,Z 778.443,A -85,B 0,C 180,E1 -1109,E2 -1109} C_VEL
LIN {X 0,Y 594.356,Z 778.444,A -85,B 0,C 180,E1 -1111.643,E2 -1111.643} C_VEL
LIN {X 0,Y 594.345,Z 778.451,A -85,B 0,C 180,E1 -1114.582,E2 -1114.582} C_VEL
LIN {X 0,Y 594.339,Z 778.445,A -85,B 0,C 180,E1 -1117.605,E2 -1117.605} C_VEL
LIN {X 0,Y 594.346,Z 778.454,A -85,B 0,C 180,E1 -1120.569,E2 -1120.569} C_VEL
LIN {X 0,Y 594.334,Z 778.446,A -85,B 0,C 180,E1 -1123.303,E2 -1123.303} C_VEL
LIN {X 0,Y 594.322,Z 778.451,A -85,B 0,C 180,E1 -1126.165,E2 -1126.165} C_VEL
LIN {X 0,Y 594.347,Z 778.448,A -85,B 0,C 180,E1 -1129.182,E2 -1129.182} C_VEL
LIN {X 0,Y 594.332,Z 778.448,A -85,B 0,C 180,E1 -1132.057,E2 -1132.057} C_VEL
LIN {X 0,Y 594.334,Z 778.47,A -85,B 0,C 180,E1 -1133.586,E2 -1133.586} C_VEL
LIN {X 0,Y 595.042,Z 783.658,A -85,B 0,C 180,E1 -1134.64,E2 -1134.64} C_VEL
LIN {X 0,Y 594.942,Z 797.463,A -85,B 0,C 180,E1 -1137.489,E2 -1137.489} C_VEL
LIN {X 0,Y 594.817,Z 811.157,A -85,B 0,C 180,E1 -1140.25,E2 -1140.25} C_VEL
LIN {X 0,Y 594.716,Z 824.852,A -85,B 0,C 180,E1 -1142.939,E2 -1142.939} C_VEL
LIN {X 0,Y 594.666,Z 838.547,A -85,B 0,C 180,E1 -1145.568,E2 -1145.568} C_VEL
LIN {X 0,Y 594.524,Z 852.242,A -85,B 0,C 180,E1 -1148.14,E2 -1148.14} C_VEL
LIN {X 0,Y 594.49,Z 865.936,A -85,B 0,C 180,E1 -1150.671,E2 -1150.671} C_VEL
LIN {X 0,Y 594.437,Z 881.587,A -85,B 0,C 180,E1 -1153.517,E2 -1153.517} C_VEL
LIN {X 0,Y 594.357,Z 897.238,A -85,B 0,C 180,E1 -1156.322,E2 -1156.322} C_VEL
LIN {X 0,Y 594.347,Z 906.189,A -85,B 0,C 180,E1 -1157.907,E2 -1157.907} C_VEL
LIN {X 0,Y 594.663,Z 912.021,A -85,B 0,C 180,E1 -1158,E2 -1158} C_VEL
LIN {X 0,Y 594.623,Z 925.265,A -85,B 0,C 180,E1 -1158.302,E2 -1158.302} C_VEL
LIN {X 0,Y 594.568,Z 938.443,A -85,B 0,C 180,E1 -1158.752,E2 -1158.752} C_VEL
LIN {X 0,Y 594.545,Z 949.66,A -85,B 0,C 180,E1 -1159.272,E2 -1159.272} C_VEL
LIN {X 0,Y 594.464,Z 961.219,A -85,B 0,C 180,E1 -1159.959,E2 -1159.959} C_VEL
LIN {X 0,Y 594.414,Z 971.612,A -85,B 0,C 180,E1 -1160.731,E2 -1160.731} C_VEL
LIN {X 0,Y 594.348,Z 980.029,A -85,B 0,C 180,E1 -1161.501,E2 -1161.501} C_VEL
LIN {X 0,Y 594.346,Z 987.972,A -85,B 0,C 180,E1 -1162.357,E2 -1162.357} C_VEL
LIN {X 0,Y 594.279,Z 995.83,A -85,B 0,C 180,E1 -1163.411,E2 -1163.411} C_VEL
LIN {X 0,Y 594.289,Z 1002.687,A -85,B 0,C 180,E1 -1164.573,E2 -1164.573} C_VEL
LIN {X 0,Y 594.27,Z 1007.376,A -85,B 0,C 180,E1 -1165.593,E2 -1165.593} C_VEL
LIN {X 0,Y 594.267,Z 1010.96,A -85,B 0,C 180,E1 -1166.611,E2 -1166.611} C_VEL
LIN {X 0,Y 594.226,Z 1012.812,A -85,B 0,C 180,E1 -1167.29,E2 -1167.29} C_VEL
LIN {X 0,Y 594.24,Z 1014.204,A -85,B 0,C 180,E1 -1167.968,E2 -1167.968} C_VEL
LIN {X 0,Y 594.239,Z 1015.785,A -85,B 0,C 180,E1 -1169.324,E2 -1169.324} C_VEL
LIN {X 0,Y 594.236,Z 1016,A -85,B 0,C 180,E1 -1170.001,E2 -1170.001} C_VEL
LIN {X 0,Y 594.247,Z 1015.183,A -85,B 0,C 180,E1 -1171.357,E2 -1171.357} C_VEL
LIN {X 0,Y 594.24,Z 1014.2,A -85,B 0,C 180,E1 -1172.034,E2 -1172.034} C_VEL
LIN {X 0,Y 594.226,Z 1012.806,A -85,B 0,C 180,E1 -1172.713,E2 -1172.713} C_VEL
LIN {X 0,Y 594.289,Z 1009.892,A -85,B 0,C 180,E1 -1173.73,E2 -1173.73} C_VEL
LIN {X 0,Y 594.241,Z 1005.945,A -85,B 0,C 180,E1 -1174.75,E2 -1174.75} C_VEL
LIN {X 0,Y 594.304,Z 999.87,A -85,B 0,C 180,E1 -1175.94,E2 -1175.94} C_VEL
LIN {X 0,Y 594.309,Z 993.228,A -85,B 0,C 180,E1 -1176.963,E2 -1176.963} C_VEL
LIN {X 0,Y 594.36,Z 984.98,A -85,B 0,C 180,E1 -1177.987,E2 -1177.987} C_VEL
LIN {X 0,Y 594.405,Z 974.587,A -85,B 0,C 180,E1 -1179.014,E2 -1179.014} C_VEL
LIN {X 0,Y 594.452,Z 963.732,A -85,B 0,C 180,E1 -1179.872,E2 -1179.872} C_VEL
LIN {X 0,Y 594.526,Z 952.755,A -85,B 0,C 180,E1 -1180.559,E2 -1180.559} C_VEL
LIN {X 0,Y 594.56,Z 940.623,A -85,B 0,C 180,E1 -1181.156,E2 -1181.156} C_VEL
LIN {X 0,Y 594.619,Z 928.847,A -85,B 0,C 180,E1 -1181.592,E2 -1181.592} C_VEL
LIN {X 0,Y 594.643,Z 916.457,A -85,B 0,C 180,E1 -1181.916,E2 -1181.916} C_VEL
LIN {X 0,Y 594.405,Z 906.586,A -85,B 0,C 180,E1 -1182.086,E2 -1182.086} C_VEL
LIN {X 0,Y 594.354,Z 906.028,A -85,B 0,C 180,E1 -1182.117,E2 -1182.117} C_VEL
LIN {X 0,Y 594.37,Z 889.399,A -85,B 0,C 180,E1 -1185.079,E2 -1185.079} C_VEL
LIN {X 0,Y 594.458,Z 875.704,A -85,B 0,C 180,E1 -1187.547,E2 -1187.547} C_VEL
LIN {X 0,Y 594.483,Z 863.966,A -85,B 0,C 180,E1 -1189.691,E2 -1189.691} C_VEL
LIN {X 0,Y 594.635,Z 847.213,A -85,B 0,C 180,E1 -1192.797,E2 -1192.797} C_VEL
LIN {X 0,Y 594.698,Z 832.664,A -85,B 0,C 180,E1 -1195.554,E2 -1195.554} C_VEL
LIN {X 0,Y 594.776,Z 817.013,A -85,B 0,C 180,E1 -1198.592,E2 -1198.592} C_VEL
LIN {X 0,Y 594.9,Z 803.318,A -85,B 0,C 180,E1 -1201.32,E2 -1201.32} C_VEL
LIN {X 0,Y 594.998,Z 789.166,A -85,B 0,C 180,E1 -1204.226,E2 -1204.226} C_VEL
LIN {X 0,Y 594.924,Z 781.516,A -85,B 0,C 180,E1 -1205.786,E2 -1205.786} C_VEL
LIN {X 0,Y 594.34,Z 778.453,A -85,B 0,C 180,E1 -1206.445,E2 -1206.445} C_VEL
LIN {X 0,Y 594.321,Z 778.452,A -85,B 0,C 180,E1 -1208.811,E2 -1208.811} C_VEL
LIN {X 0,Y 594.338,Z 778.449,A -85,B 0,C 180,E1 -1211.843,E2 -1211.843} C_VEL
LIN {X 0,Y 594.336,Z 778.446,A -85,B 0,C 180,E1 -1214.241,E2 -1214.241} C_VEL
LIN {X 0,Y 594.318,Z 778.452,A -85,B 0,C 180,E1 -1217.154,E2 -1217.154} C_VEL
LIN {X 0,Y 594.323,Z 778.455,A -85,B 0,C 180,E1 -1219.429,E2 -1219.429} C_VEL
LIN {X 0,Y 594.301,Z 778.455,A -85,B 0,C 180,E1 -1222.053,E2 -1222.053} C_VEL
LIN {X 0,Y 594.295,Z 778.45,A -85,B 0,C 180,E1 -1224.685,E2 -1224.685} C_VEL
LIN {X 0,Y 594.336,Z 778.446,A -85,B 0,C 180,E1 -1227.096,E2 -1227.096} C_VEL
LIN {X 0,Y 594.365,Z 778.448,A -85,B 0,C 180,E1 -1229.676,E2 -1229.676} C_VEL
LIN {X 0,Y 594.319,Z 778.45,A -85,B 0,C 180,E1 -1232.536,E2 -1232.536} C_VEL
LIN {X 0,Y 594.316,Z 778.449,A -85,B 0,C 180,E1 -1234.804,E2 -1234.804} C_VEL
LIN {X 0,Y 594.303,Z 778.449,A -85,B 0,C 180,E1 -1237.28,E2 -1237.28} C_VEL
LIN {X 0,Y 594.333,Z 778.451,A -85,B 0,C 180,E1 -1239.945,E2 -1239.945} C_VEL
LIN {X 0,Y 594.315,Z 778.452,A -85,B 0,C 180,E1 -1242.804,E2 -1242.804} C_VEL
LIN {X 0,Y 594.328,Z 778.447,A -85,B 0,C 180,E1 -1245.621,E2 -1245.621} C_VEL
LIN {X 0,Y 594.41,Z 778.542,A -85,B 0,C 180,E1 -1248.439,E2 -1248.439} C_VEL
LIN {X 0,Y 594.503,Z 790.248,A -85,B 0,C 180,E1 -1248.873,E2 -1248.873} C_VEL
LIN {X 0,Y 594.417,Z 801.928,A -85,B 0,C 180,E1 -1249.44,E2 -1249.44} C_VEL
LIN {X 0,Y 594.413,Z 813.069,A -85,B 0,C 180,E1 -1250.128,E2 -1250.128} C_VEL
LIN {X 0,Y 594.396,Z 823.123,A -85,B 0,C 180,E1 -1250.901,E2 -1250.901} C_VEL
LIN {X 0,Y 594.362,Z 832.973,A -85,B 0,C 180,E1 -1251.843,E2 -1251.843} C_VEL
LIN {X 0,Y 594.317,Z 840.332,A -85,B 0,C 180,E1 -1252.697,E2 -1252.697} C_VEL
LIN {X 0,Y 594.296,Z 846.919,A -85,B 0,C 180,E1 -1253.623,E2 -1253.623} C_VEL
LIN {X 0,Y 594.289,Z 852.433,A -85,B 0,C 180,E1 -1254.571,E2 -1254.571} C_VEL
LIN {X 0,Y 594.27,Z 857.172,A -85,B 0,C 180,E1 -1255.591,E2 -1255.591} C_VEL
LIN {X 0,Y 594.268,Z 860.807,A -85,B 0,C 180,E1 -1256.61,E2 -1256.61} C_VEL
LIN {X 0,Y 594.225,Z 862.694,A -85,B 0,C 180,E1 -1257.288,E2 -1257.288} C_VEL
LIN {X 0,Y 594.24,Z 864.13,A -85,B 0,C 180,E1 -1257.967,E2 -1257.967} C_VEL
LIN {X 0,Y 594.24,Z 865.753,A -85,B 0,C 180,E1 -1259.322,E2 -1259.322} C_VEL
LIN {X 0,Y 594.236,Z 865.996,A -85,B 0,C 180,E1 -1260,E2 -1260} C_VEL
LIN {X 0,Y 594.239,Z 865.815,A -85,B 0,C 180,E1 -1260.678,E2 -1260.678} C_VEL
LIN {X 0,Y 594.239,Z 864.276,A -85,B 0,C 180,E1 -1262.033,E2 -1262.033} C_VEL
LIN {X 0,Y 594.226,Z 862.901,A -85,B 0,C 180,E1 -1262.712,E2 -1262.712} C_VEL
LIN {X 0,Y 594.289,Z 860.026,A -85,B 0,C 180,E1 -1263.729,E2 -1263.729} C_VEL
LIN {X 0,Y 594.241,Z 856.127,A -85,B 0,C 180,E1 -1264.749,E2 -1264.749} C_VEL
LIN {X 0,Y 594.299,Z 851.1,A -85,B 0,C 180,E1 -1265.769,E2 -1265.769} C_VEL
LIN {X 0,Y 594.317,Z 844.786,A -85,B 0,C 180,E1 -1266.791,E2 -1266.791} C_VEL
LIN {X 0,Y 594.347,Z 836.868,A -85,B 0,C 180,E1 -1267.816,E2 -1267.816} C_VEL
LIN {X 0,Y 594.368,Z 826.996,A -85,B 0,C 180,E1 -1268.842,E2 -1268.842} C_VEL
LIN {X 0,Y 594.44,Z 816.703,A -85,B 0,C 180,E1 -1269.699,E2 -1269.699} C_VEL
LIN {X 0,Y 594.436,Z 805.089,A -85,B 0,C 180,E1 -1270.473,E2 -1270.473} C_VEL
LIN {X 0,Y 594.484,Z 794.135,A -85,B 0,C 180,E1 -1271.046,E2 -1271.046} C_VEL
LIN {X 0,Y 594.554,Z 782.914,A -85,B 0,C 180,E1 -1271.501,E2 -1271.501} C_VEL
LIN {X 0,Y 594.288,Z 780.936,A -85,B 0,C 180,E1 -1271.642,E2 -1271.642} C_VEL
LIN {X 0,Y 593.454,Z 779.401,A -85,B 0,C 180,E1 -1271.926,E2 -1271.926} C_VEL
LIN {X 0,Y 592.035,Z 778.796,A -85,B 0,C 180,E1 -1272.356,E2 -1272.356} C_VEL
LIN {X 0,Y 588.401,Z 779.226,A -85,B 0,C 180,E1 -1273.567,E2 -1273.567} C_VEL
LIN {X 0,Y 587.377,Z 779.318,A -85,B 0,C 180,E1 -1274.224,E2 -1274.224} C_VEL
LIN {X 0,Y 587.301,Z 779.322,A -85,B 0,C 180,E1 -1274.446,E2 -1274.446} C_VEL
LIN {X 0,Y 587.263,Z 779.334,A -85,B 0,C 180,E1 -1277.409,E2 -1277.409} C_VEL
LIN {X 0,Y 587.28,Z 779.325,A -85,B 0,C 180,E1 -1280.307,E2 -1280.307} C_VEL
LIN {X 0,Y 587.287,Z 779.327,A -85,B 0,C 180,E1 -1283.26,E2 -1283.26} C_VEL
LIN {X 0,Y 587.306,Z 779.324,A -85,B 0,C 180,E1 -1286.169,E2 -1286.169} C_VEL
LIN {X 0,Y 587.3,Z 779.323,A -85,B 0,C 180,E1 -1289.124,E2 -1289.124} C_VEL
LIN {X 0,Y 587.319,Z 779.33,A -85,B 0,C 180,E1 -1291.831,E2 -1291.831} C_VEL
LIN {X 0,Y 587.33,Z 779.321,A -85,B 0,C 180,E1 -1294.344,E2 -1294.344} C_VEL
LIN {X 0,Y 587.317,Z 779.325,A -85,B 0,C 180,E1 -1297.61,E2 -1297.61} C_VEL
LIN {X 0,Y 587.306,Z 779.327,A -85,B 0,C 180,E1 -1300.255,E2 -1300.255} C_VEL
LIN {X 0,Y 587.294,Z 779.322,A -85,B 0,C 180,E1 -1303.009,E2 -1303.009} C_VEL
LIN {X 0,Y 587.319,Z 779.33,A -85,B 0,C 180,E1 -1306.048,E2 -1306.048} C_VEL
LIN {X 0,Y 587.337,Z 779.318,A -85,B 0,C 180,E1 -1308.925,E2 -1308.925} C_VEL
LIN {X 0,Y 587.32,Z 779.321,A -85,B 0,C 180,E1 -1311.519,E2 -1311.519} C_VEL
LIN {X 0,Y 587.292,Z 779.332,A -85,B 0,C 180,E1 -1314.099,E2 -1314.099} C_VEL
LIN {X 0,Y 587.34,Z 779.318,A -85,B 0,C 180,E1 -1316.889,E2 -1316.889} C_VEL
LIN {X 0,Y 587.326,Z 779.319,A -85,B 0,C 180,E1 -1319.493,E2 -1319.493} C_VEL
LIN {X 0,Y 587.347,Z 779.327,A -85,B 0,C 180,E1 -1322.309,E2 -1322.309} C_VEL
LIN {X 0,Y 587.32,Z 779.319,A -85,B 0,C 180,E1 -1325.239,E2 -1325.239} C_VEL
LIN {X 0,Y 587.342,Z 779.317,A -85,B 0,C 180,E1 -1327.485,E2 -1327.485} C_VEL
LIN {X 0,Y 587.329,Z 779.319,A -85,B 0,C 180,E1 -1329.694,E2 -1329.694} C_VEL
LIN {X 0,Y 587.303,Z 779.324,A -85,B 0,C 180,E1 -1331.872,E2 -1331.872} C_VEL
LIN {X 0,Y 587.323,Z 779.323,A -85,B 0,C 180,E1 -1334.024,E2 -1334.024} C_VEL
LIN {X 0,Y 587.354,Z 779.32,A -85,B 0,C 180,E1 -1336.153,E2 -1336.153} C_VEL
LIN {X 0,Y 587.376,Z 779.501,A -85,B 0,C 180,E1 -1338.333,E2 -1338.333} C_VEL
LIN {X 0,Y 587.618,Z 785.539,A -85,B 0,C 180,E1 -1338.548,E2 -1338.548} C_VEL
LIN {X 0,Y 587.558,Z 798.723,A -85,B 0,C 180,E1 -1339.14,E2 -1339.14} C_VEL
LIN {X 0,Y 587.444,Z 809.173,A -85,B 0,C 180,E1 -1339.748,E2 -1339.748} C_VEL
LIN {X 0,Y 587.392,Z 818.862,A -85,B 0,C 180,E1 -1340.443,E2 -1340.443} C_VEL
LIN {X 0,Y 587.338,Z 827.833,A -85,B 0,C 180,E1 -1341.223,E2 -1341.223} C_VEL
LIN {X 0,Y 587.288,Z 836.064,A -85,B 0,C 180,E1 -1342.089,E2 -1342.089} C_VEL
LIN {X 0,Y 587.232,Z 844.127,A -85,B 0,C 180,E1 -1343.125,E2 -1343.125} C_VEL
LIN {X 0,Y 587.237,Z 850.607,A -85,B 0,C 180,E1 -1344.16,E2 -1344.16} C_VEL
LIN {X 0,Y 587.146,Z 855.752,A -85,B 0,C 180,E1 -1345.192,E2 -1345.192} C_VEL
LIN {X 0,Y 587.212,Z 859.741,A -85,B 0,C 180,E1 -1346.225,E2 -1346.225} C_VEL
LIN {X 0,Y 587.131,Z 862.691,A -85,B 0,C 180,E1 -1347.254,E2 -1347.254} C_VEL
LIN {X 0,Y 587.146,Z 865.131,A -85,B 0,C 180,E1 -1348.627,E2 -1348.627} C_VEL
LIN {X 0,Y 587.14,Z 865.753,A -85,B 0,C 180,E1 -1349.313,E2 -1349.313} C_VEL
LIN {X 0,Y 587.14,Z 865.816,A -85,B 0,C 180,E1 -1350.685,E2 -1350.685} C_VEL
LIN {X 0,Y 587.139,Z 864.274,A -85,B 0,C 180,E1 -1352.057,E2 -1352.057} C_VEL
LIN {X 0,Y 587.132,Z 862.918,A -85,B 0,C 180,E1 -1352.743,E2 -1352.743} C_VEL
LIN {X 0,Y 587.213,Z 860.044,A -85,B 0,C 180,E1 -1353.773,E2 -1353.773} C_VEL
LIN {X 0,Y 587.147,Z 856.146,A -85,B 0,C 180,E1 -1354.805,E2 -1354.805} C_VEL
LIN {X 0,Y 587.229,Z 851.117,A -85,B 0,C 180,E1 -1355.837,E2 -1355.837} C_VEL
LIN {X 0,Y 587.229,Z 844.788,A -85,B 0,C 180,E1 -1356.872,E2 -1356.872} C_VEL
LIN {X 0,Y 587.273,Z 836.859,A -85,B 0,C 180,E1 -1357.909,E2 -1357.909} C_VEL
LIN {X 0,Y 587.324,Z 828.791,A -85,B 0,C 180,E1 -1358.774,E2 -1358.774} C_VEL
LIN {X 0,Y 587.392,Z 820.016,A -85,B 0,C 180,E1 -1359.555,E2 -1359.555} C_VEL
LIN {X 0,Y 587.439,Z 810.561,A -85,B 0,C 180,E1 -1360.25,E2 -1360.25} C_VEL
LIN {X 0,Y 587.543,Z 800.417,A -85,B 0,C 180,E1 -1360.858,E2 -1360.858} C_VEL
LIN {X 0,Y 587.598,Z 788.224,A -85,B 0,C 180,E1 -1361.436,E2 -1361.436} C_VEL
LIN {X 0,Y 587.393,Z 779.517,A -85,B 0,C 180,E1 -1361.756,E2 -1361.756} C_VEL
LIN {X 0,Y 587.339,Z 779.318,A -85,B 0,C 180,E1 -1364.552,E2 -1364.552} C_VEL
LIN {X 0,Y 587.348,Z 779.322,A -85,B 0,C 180,E1 -1367.404,E2 -1367.404} C_VEL
LIN {X 0,Y 587.327,Z 779.321,A -85,B 0,C 180,E1 -1370.303,E2 -1370.303} C_VEL
LIN {X 0,Y 587.321,Z 779.321,A -85,B 0,C 180,E1 -1373.257,E2 -1373.257} C_VEL
LIN {X 0,Y 587.331,Z 779.323,A -85,B 0,C 180,E1 -1375.515,E2 -1375.515} C_VEL
LIN {X 0,Y 587.345,Z 779.325,A -85,B 0,C 180,E1 -1377.816,E2 -1377.816} C_VEL
LIN {X 0,Y 587.338,Z 779.32,A -85,B 0,C 180,E1 -1380.509,E2 -1380.509} C_VEL
LIN {X 0,Y 587.329,Z 779.319,A -85,B 0,C 180,E1 -1383.395,E2 -1383.395} C_VEL
LIN {X 0,Y 587.312,Z 779.327,A -85,B 0,C 180,E1 -1385.896,E2 -1385.896} C_VEL
LIN {X 0,Y 587.327,Z 779.324,A -85,B 0,C 180,E1 -1388.477,E2 -1388.477} C_VEL
LIN {X 0,Y 587.331,Z 779.318,A -85,B 0,C 180,E1 -1391.155,E2 -1391.155} C_VEL
LIN {X 0,Y 587.324,Z 779.326,A -85,B 0,C 180,E1 -1394.113,E2 -1394.113} C_VEL
LIN {X 0,Y 587.312,Z 779.322,A -85,B 0,C 180,E1 -1396.993,E2 -1396.993} C_VEL
LIN {X 0,Y 587.317,Z 779.32,A -85,B 0,C 180,E1 -1399.746,E2 -1399.746} C_VEL
LIN {X 0,Y 587.335,Z 779.325,A -85,B 0,C 180,E1 -1402.391,E2 -1402.391} C_VEL
LIN {X 0,Y 587.335,Z 779.322,A -85,B 0,C 180,E1 -1404.945,E2 -1404.945} C_VEL
LIN {X 0,Y 587.327,Z 779.319,A -85,B 0,C 180,E1 -1407.42,E2 -1407.42} C_VEL
LIN {X 0,Y 587.334,Z 779.317,A -85,B 0,C 180,E1 -1409.83,E2 -1409.83} C_VEL
LIN {X 0,Y 587.336,Z 779.32,A -85,B 0,C 180,E1 -1412.306,E2 -1412.306} C_VEL
LIN {X 0,Y 587.328,Z 779.323,A -85,B 0,C 180,E1 -1414.483,E2 -1414.483} C_VEL
LIN {X 0,Y 587.324,Z 779.321,A -85,B 0,C 180,E1 -1417.485,E2 -1417.485} C_VEL
LIN {X 0,Y 587.328,Z 779.32,A -85,B 0,C 180,E1 -1420.424,E2 -1420.424} C_VEL
LIN {X 0,Y 587.327,Z 779.324,A -85,B 0,C 180,E1 -1423.31,E2 -1423.31} C_VEL
LIN {X 0,Y 587.344,Z 779.316,A -85,B 0,C 180,E1 -1426.154,E2 -1426.154} C_VEL
LIN {X 0,Y 587.395,Z 779.317,A -85,B 0,C 180,E1 -1428.963,E2 -1428.963} C_VEL
LIN {X 0,Y 587.35,Z 779.319,A -85,B 0,C 180,E1 -1431.744,E2 -1431.744} C_VEL
LIN {X 0,Y 587.344,Z 779.317,A -85,B 0,C 180,E1 -1434.507,E2 -1434.507} C_VEL
LIN {X 0,Y 587.373,Z 779.321,A -85,B 0,C 180,E1 -1437.257,E2 -1437.257} C_VEL
LIN {X 0,Y 587.351,Z 779.318,A -85,B 0,C 180,E1 -1440,E2 -1440} C_VEL
LIN {X 0,Y 587.349,Z 779.316,A -85,B 0,C 180,E1 -1442.743,E2 -1442.743} C_VEL
LIN {X 0,Y 587.349,Z 779.325,A -85,B 0,C 180,E1 -1445.493,E2 -1445.493} C_VEL
LIN {X 0,Y 587.343,Z 779.318,A -85,B 0,C 180,E1 -1448.256,E2 -1448.256} C_VEL
LIN {X 0,Y 587.329,Z 779.32,A -85,B 0,C 180,E1 -1451.134,E2 -1451.134} C_VEL
LIN {X 0,Y 587.322,Z 779.323,A -85,B 0,C 180,E1 -1454.252,E2 -1454.252} C_VEL
LIN {X 0,Y 587.33,Z 779.321,A -85,B 0,C 180,E1 -1457.407,E2 -1457.407} C_VEL
LIN {X 0,Y 587.301,Z 779.327,A -85,B 0,C 180,E1 -1460.306,E2 -1460.306} C_VEL
LIN {X 0,Y 587.298,Z 779.322,A -85,B 0,C 180,E1 -1463.26,E2 -1463.26} C_VEL
LIN {X 0,Y 587.308,Z 779.322,A -85,B 0,C 180,E1 -1465.518,E2 -1465.518} C_VEL
LIN {X 0,Y 587.297,Z 779.326,A -85,B 0,C 180,E1 -1468.598,E2 -1468.598} C_VEL
LIN {X 0,Y 587.309,Z 779.322,A -85,B 0,C 180,E1 -1470.968,E2 -1470.968} C_VEL
LIN {X 0,Y 587.309,Z 779.321,A -85,B 0,C 180,E1 -1473.398,E2 -1473.398} C_VEL
LIN {X 0,Y 587.262,Z 779.33,A -85,B 0,C 180,E1 -1475.902,E2 -1475.902} C_VEL
LIN {X 0,Y 587.298,Z 779.333,A -85,B 0,C 180,E1 -1478.482,E2 -1478.482} C_VEL
LIN {X 0,Y 587.288,Z 779.325,A -85,B 0,C 180,E1 -1481.161,E2 -1481.161} C_VEL
LIN {X 0,Y 587.282,Z 779.326,A -85,B 0,C 180,E1 -1483.955,E2 -1483.955} C_VEL
LIN {X 0,Y 587.264,Z 779.332,A -85,B 0,C 180,E1 -1486.991,E2 -1486.991} C_VEL
LIN {X 0,Y 587.28,Z 779.325,A -85,B 0,C 180,E1 -1489.745,E2 -1489.745} C_VEL
LIN {X 0,Y 587.318,Z 779.326,A -85,B 0,C 180,E1 -1492.393,E2 -1492.393} C_VEL
LIN {X 0,Y 587.325,Z 779.449,A -85,B 0,C 180,E1 -1493.397,E2 -1493.397} C_VEL
LIN {X 0,Y 588.101,Z 784.049,A -85,B 0,C 180,E1 -1494.353,E2 -1494.353} C_VEL
LIN {X 0,Y 588.172,Z 793.55,A -85,B 0,C 180,E1 -1496.248,E2 -1496.248} C_VEL
LIN {X 0,Y 588.017,Z 807.245,A -85,B 0,C 180,E1 -1499.076,E2 -1499.076} C_VEL
LIN {X 0,Y 587.823,Z 820.939,A -85,B 0,C 180,E1 -1501.821,E2 -1501.821} C_VEL
LIN {X 0,Y 587.764,Z 834.634,A -85,B 0,C 180,E1 -1504.505,E2 -1504.505} C_VEL
LIN {X 0,Y 587.648,Z 849.115,A -85,B 0,C 180,E1 -1507.278,E2 -1507.278} C_VEL
LIN {X 0,Y 587.505,Z 865.936,A -85,B 0,C 180,E1 -1510.432,E2 -1510.432} C_VEL
LIN {X 0,Y 587.424,Z 881.587,A -85,B 0,C 180,E1 -1513.315,E2 -1513.315} C_VEL
LIN {X 0,Y 587.302,Z 897.238,A -85,B 0,C 180,E1 -1516.154,E2 -1516.154} C_VEL
LIN {X 0,Y 587.309,Z 906.189,A -85,B 0,C 180,E1 -1517.76,E2 -1517.76} C_VEL
LIN {X 0,Y 587.737,Z 912.021,A -85,B 0,C 180,E1 -1517.857,E2 -1517.857} C_VEL
LIN {X 0,Y 587.673,Z 925.264,A -85,B 0,C 180,E1 -1518.162,E2 -1518.162} C_VEL
LIN {X 0,Y 587.604,Z 937.85,A -85,B 0,C 180,E1 -1518.594,E2 -1518.594} C_VEL
LIN {X 0,Y 587.56,Z 949.659,A -85,B 0,C 180,E1 -1519.143,E2 -1519.143} C_VEL
LIN {X 0,Y 587.444,Z 961.22,A -85,B 0,C 180,E1 -1519.838,E2 -1519.838} C_VEL
LIN {X 0,Y 587.366,Z 971.613,A -85,B 0,C 180,E1 -1520.619,E2 -1520.619} C_VEL
LIN {X 0,Y 587.298,Z 980.037,A -85,B 0,C 180,E1 -1521.399,E2 -1521.399} C_VEL
LIN {X 0,Y 587.273,Z 987.972,A -85,B 0,C 180,E1 -1522.264,E2 -1522.264} C_VEL
LIN {X 0,Y 587.229,Z 994.48,A -85,B 0,C 180,E1 -1523.128,E2 -1523.128} C_VEL
LIN {X 0,Y 587.236,Z 1000.873,A -85,B 0,C 180,E1 -1524.163,E2 -1524.163} C_VEL
LIN {X 0,Y 587.147,Z 1005.955,A -85,B 0,C 180,E1 -1525.195,E2 -1525.195} C_VEL
LIN {X 0,Y 587.212,Z 1009.9,A -85,B 0,C 180,E1 -1526.227,E2 -1526.227} C_VEL
LIN {X 0,Y 587.132,Z 1012.813,A -85,B 0,C 180,E1 -1527.257,E2 -1527.257} C_VEL
LIN {X 0,Y 587.139,Z 1014.204,A -85,B 0,C 180,E1 -1527.943,E2 -1527.943} C_VEL
LIN {X 0,Y 587.14,Z 1015.785,A -85,B 0,C 180,E1 -1529.315,E2 -1529.315} C_VEL
LIN {X 0,Y 587.137,Z 1016,A -85,B 0,C 180,E1 -1530.001,E2 -1530.001} C_VEL
LIN {X 0,Y 587.147,Z 1015.183,A -85,B 0,C 180,E1 -1531.373,E2 -1531.373} C_VEL
LIN {X 0,Y 587.139,Z 1014.199,A -85,B 0,C 180,E1 -1532.059,E2 -1532.059} C_VEL
LIN {X 0,Y 587.132,Z 1012.806,A -85,B 0,C 180,E1 -1532.746,E2 -1532.746} C_VEL
LIN {X 0,Y 587.213,Z 1009.892,A -85,B 0,C 180,E1 -1533.775,E2 -1533.775} C_VEL
LIN {X 0,Y 587.147,Z 1005.945,A -85,B 0,C 180,E1 -1534.808,E2 -1534.808} C_VEL
LIN {X 0,Y 587.217,Z 999.87,A -85,B 0,C 180,E1 -1536.012,E2 -1536.012} C_VEL
LIN {X 0,Y 587.246,Z 993.228,A -85,B 0,C 180,E1 -1537.047,E2 -1537.047} C_VEL
LIN {X 0,Y 587.298,Z 984.98,A -85,B 0,C 180,E1 -1538.084,E2 -1538.084} C_VEL
LIN {X 0,Y 587.358,Z 974.587,A -85,B 0,C 180,E1 -1539.123,E2 -1539.123} C_VEL
LIN {X 0,Y 587.433,Z 964.916,A -85,B 0,C 180,E1 -1539.904,E2 -1539.904} C_VEL
LIN {X 0,Y 587.528,Z 954.309,A -85,B 0,C 180,E1 -1540.599,E2 -1540.599} C_VEL
LIN {X 0,Y 587.578,Z 941.642,A -85,B 0,C 180,E1 -1541.245,E2 -1541.245} C_VEL
LIN {X 0,Y 587.683,Z 928.847,A -85,B 0,C 180,E1 -1541.731,E2 -1541.731} C_VEL
LIN {X 0,Y 587.715,Z 916.456,A -85,B 0,C 180,E1 -1542.059,E2 -1542.059} C_VEL
LIN {X 0,Y 587.499,Z 907.528,A -85,B 0,C 180,E1 -1542.216,E2 -1542.216} C_VEL
LIN {X 0,Y 587.316,Z 906.028,A -85,B 0,C 180,E1 -1542.264,E2 -1542.264} C_VEL
LIN {X 0,Y 587.355,Z 889.399,A -85,B 0,C 180,E1 -1545.263,E2 -1545.263} C_VEL
LIN {X 0,Y 587.452,Z 875.704,A -85,B 0,C 180,E1 -1547.763,E2 -1547.763} C_VEL
LIN {X 0,Y 587.501,Z 862.01,A -85,B 0,C 180,E1 -1550.3,E2 -1550.3} C_VEL
LIN {X 0,Y 587.644,Z 846.358,A -85,B 0,C 180,E1 -1553.246,E2 -1553.246} C_VEL
LIN {X 0,Y 587.767,Z 832.664,A -85,B 0,C 180,E1 -1555.878,E2 -1555.878} C_VEL
LIN {X 0,Y 587.858,Z 818.969,A -85,B 0,C 180,E1 -1558.57,E2 -1558.57} C_VEL
LIN {X 0,Y 588.049,Z 805.274,A -85,B 0,C 180,E1 -1561.325,E2 -1561.325} C_VEL
LIN {X 0,Y 588.177,Z 791.558,A -85,B 0,C 180,E1 -1564.167,E2 -1564.167} C_VEL
LIN {X 0,Y 588.014,Z 783.059,A -85,B 0,C 180,E1 -1565.85,E2 -1565.85} C_VEL
LIN {X 0,Y 587.306,Z 779.33,A -85,B 0,C 180,E1 -1566.639,E2 -1566.639} C_VEL
LIN {X 0,Y 587.298,Z 779.333,A -85,B 0,C 180,E1 -1569.364,E2 -1569.364} C_VEL
LIN {X 0,Y 587.288,Z 779.325,A -85,B 0,C 180,E1 -1572.102,E2 -1572.102} C_VEL
LIN {X 0,Y 587.26,Z 779.33,A -85,B 0,C 180,E1 -1574.918,E2 -1574.918} C_VEL
LIN {X 0,Y 587.301,Z 779.327,A -85,B 0,C 180,E1 -1577.923,E2 -1577.923} C_VEL
LIN {X 0,Y 587.295,Z 779.322,A -85,B 0,C 180,E1 -1580.636,E2 -1580.636} C_VEL
LIN {X 0,Y 587.264,Z 779.33,A -85,B 0,C 180,E1 -1583.304,E2 -1583.304} C_VEL
LIN {X 0,Y 587.313,Z 779.331,A -85,B 0,C 180,E1 -1585.777,E2 -1585.777} C_VEL
LIN {X 0,Y 587.302,Z 779.327,A -85,B 0,C 180,E1 -1588.229,E2 -1588.229} C_VEL
LIN {X 0,Y 587.295,Z 779.323,A -85,B 0,C 180,E1 -1590.877,E2 -1590.877} C_VEL
LIN {X 0,Y 587.295,Z 779.329,A -85,B 0,C 180,E1 -1593.833,E2 -1593.833} C_VEL
LIN {X 0,Y 587.285,Z 779.326,A -85,B 0,C 180,E1 -1596.74,E2 -1596.74} C_VEL
LIN {X 0,Y 587.282,Z 779.326,A -85,B 0,C 180,E1 -1599.693,E2 -1599.693} C_VEL
LIN {X 0,Y 587.264,Z 779.334,A -85,B 0,C 180,E1 -1602.591,E2 -1602.591} C_VEL
LIN {X 0,Y 587.299,Z 779.323,A -85,B 0,C 180,E1 -1605.446,E2 -1605.446} C_VEL
LIN {X 0,Y 587.349,Z 779.467,A -85,B 0,C 180,E1 -1608.329,E2 -1608.329} C_VEL
LIN {X 0,Y 587.582,Z 787.35,A -85,B 0,C 180,E1 -1608.618,E2 -1608.618} C_VEL
LIN {X 0,Y 587.492,Z 798.77,A -85,B 0,C 180,E1 -1609.14,E2 -1609.14} C_VEL
LIN {X 0,Y 587.381,Z 809.207,A -85,B 0,C 180,E1 -1609.748,E2 -1609.748} C_VEL
LIN {X 0,Y 587.388,Z 818.889,A -85,B 0,C 180,E1 -1610.444,E2 -1610.444} C_VEL
LIN {X 0,Y 587.337,Z 827.865,A -85,B 0,C 180,E1 -1611.224,E2 -1611.224} C_VEL
LIN {X 0,Y 587.274,Z 837.576,A -85,B 0,C 180,E1 -1612.263,E2 -1612.263} C_VEL
LIN {X 0,Y 587.217,Z 845.987,A -85,B 0,C 180,E1 -1613.402,E2 -1613.402} C_VEL
LIN {X 0,Y 587.211,Z 852.433,A -85,B 0,C 180,E1 -1614.506,E2 -1614.506} C_VEL
LIN {X 0,Y 587.188,Z 857.168,A -85,B 0,C 180,E1 -1615.538,E2 -1615.538} C_VEL
LIN {X 0,Y 587.194,Z 860.805,A -85,B 0,C 180,E1 -1616.569,E2 -1616.569} C_VEL
LIN {X 0,Y 587.132,Z 862.692,A -85,B 0,C 180,E1 -1617.256,E2 -1617.256} C_VEL
LIN {X 0,Y 587.139,Z 864.132,A -85,B 0,C 180,E1 -1617.942,E2 -1617.942} C_VEL
LIN {X 0,Y 587.14,Z 865.754,A -85,B 0,C 180,E1 -1619.314,E2 -1619.314} C_VEL
LIN {X 0,Y 587.137,Z 865.996,A -85,B 0,C 180,E1 -1620,E2 -1620} C_VEL
LIN {X 0,Y 587.148,Z 865.233,A -85,B 0,C 180,E1 -1621.372,E2 -1621.372} C_VEL
LIN {X 0,Y 587.138,Z 864.276,A -85,B 0,C 180,E1 -1622.058,E2 -1622.058} C_VEL
LIN {X 0,Y 587.133,Z 862.892,A -85,B 0,C 180,E1 -1622.744,E2 -1622.744} C_VEL
LIN {X 0,Y 587.213,Z 860.018,A -85,B 0,C 180,E1 -1623.774,E2 -1623.774} C_VEL
LIN {X 0,Y 587.147,Z 856.12,A -85,B 0,C 180,E1 -1624.806,E2 -1624.806} C_VEL
LIN {X 0,Y 587.229,Z 851.094,A -85,B 0,C 180,E1 -1625.839,E2 -1625.839} C_VEL
LIN {X 0,Y 587.231,Z 844.782,A -85,B 0,C 180,E1 -1626.874,E2 -1626.874} C_VEL
LIN {X 0,Y 587.288,Z 836.863,A -85,B 0,C 180,E1 -1627.91,E2 -1627.91} C_VEL
LIN {X 0,Y 587.338,Z 826.979,A -85,B 0,C 180,E1 -1628.949,E2 -1628.949} C_VEL
LIN {X 0,Y 587.407,Z 816.698,A -85,B 0,C 180,E1 -1629.817,E2 -1629.817} C_VEL
LIN {X 0,Y 587.443,Z 805.082,A -85,B 0,C 180,E1 -1630.6,E2 -1630.6} C_VEL
LIN {X 0,Y 587.513,Z 793.367,A -85,B 0,C 180,E1 -1631.212,E2 -1631.212} C_VEL
LIN {X 0,Y 587.614,Z 781.604,A -85,B 0,C 180,E1 -1631.683,E2 -1631.683} C_VEL
LIN {X 0,Y 587.346,Z 779.324,A -85,B 0,C 180,E1 -1631.781,E2 -1631.781} C_VEL
LIN {X 0,Y 587.301,Z 779.322,A -85,B 0,C 180,E1 -1634.446,E2 -1634.446} C_VEL
LIN {X 0,Y 586.64,Z 779.408,A -85,B 0,C 180,E1 -1635.018,E2 -1635.018} C_VEL
LIN {X 0,Y 583.758,Z 779.768,A -85,B 0,C 180,E1 -1635.946,E2 -1635.946} C_VEL
LIN {X 0,Y 581.326,Z 780.069,A -85,B 0,C 180,E1 -1636.692,E2 -1636.692} C_VEL
LIN {X 0,Y 580.295,Z 780.2,A -85,B 0,C 180,E1 -1637.269,E2 -1637.269} C_VEL
LIN {X 0,Y 580.219,Z 780.212,A -85,B 0,C 180,E1 -1637.464,E2 -1637.464} C_VEL
LIN {X 0,Y 580.237,Z 780.208,A -85,B 0,C 180,E1 -1639.825,E2 -1639.825} C_VEL
LIN {X 0,Y 580.246,Z 780.2,A -85,B 0,C 180,E1 -1642.805,E2 -1642.805} C_VEL
LIN {X 0,Y 580.244,Z 780.202,A -85,B 0,C 180,E1 -1645.083,E2 -1645.083} C_VEL
LIN {X 0,Y 580.234,Z 780.211,A -85,B 0,C 180,E1 -1647.846,E2 -1647.846} C_VEL
LIN {X 0,Y 580.268,Z 780.198,A -85,B 0,C 180,E1 -1650.691,E2 -1650.691} C_VEL
LIN {X 0,Y 580.273,Z 780.198,A -85,B 0,C 180,E1 -1653.311,E2 -1653.311} C_VEL
LIN {X 0,Y 580.226,Z 780.211,A -85,B 0,C 180,E1 -1655.753,E2 -1655.753} C_VEL
LIN {X 0,Y 580.282,Z 780.203,A -85,B 0,C 180,E1 -1658.147,E2 -1658.147} C_VEL
LIN {X 0,Y 580.279,Z 780.196,A -85,B 0,C 180,E1 -1660.845,E2 -1660.845} C_VEL
LIN {X 0,Y 580.24,Z 780.203,A -85,B 0,C 180,E1 -1663.386,E2 -1663.386} C_VEL
LIN {X 0,Y 580.253,Z 780.206,A -85,B 0,C 180,E1 -1666.339,E2 -1666.339} C_VEL
LIN {X 0,Y 580.298,Z 780.194,A -85,B 0,C 180,E1 -1669.156,E2 -1669.156} C_VEL
LIN {X 0,Y 580.29,Z 780.202,A -85,B 0,C 180,E1 -1671.927,E2 -1671.927} C_VEL
LIN {X 0,Y 580.254,Z 780.206,A -85,B 0,C 180,E1 -1674.452,E2 -1674.452} C_VEL
LIN {X 0,Y 580.291,Z 780.196,A -85,B 0,C 180,E1 -1676.974,E2 -1676.974} C_VEL
LIN {X 0,Y 580.288,Z 780.195,A -85,B 0,C 180,E1 -1679.424,E2 -1679.424} C_VEL
LIN {X 0,Y 580.295,Z 780.202,A -85,B 0,C 180,E1 -1682.143,E2 -1682.143} C_VEL
LIN {X 0,Y 580.295,Z 780.196,A -85,B 0,C 180,E1 -1684.919,E2 -1684.919} C_VEL
LIN {X 0,Y 580.272,Z 780.201,A -85,B 0,C 180,E1 -1687.946,E2 -1687.946} C_VEL
LIN {X 0,Y 580.304,Z 780.198,A -85,B 0,C 180,E1 -1690.913,E2 -1690.913} C_VEL
LIN {X 0,Y 580.278,Z 780.199,A -85,B 0,C 180,E1 -1693.825,E2 -1693.825} C_VEL
LIN {X 0,Y 580.322,Z 780.194,A -85,B 0,C 180,E1 -1695.982,E2 -1695.982} C_VEL
LIN {X 0,Y 580.306,Z 780.199,A -85,B 0,C 180,E1 -1698.206,E2 -1698.206} C_VEL
LIN {X 0,Y 580.69,Z 783.913,A -85,B 0,C 180,E1 -1698.347,E2 -1698.347} C_VEL
LIN {X 0,Y 580.576,Z 797.035,A -85,B 0,C 180,E1 -1698.919,E2 -1698.919} C_VEL
LIN {X 0,Y 580.47,Z 807.852,A -85,B 0,C 180,E1 -1699.535,E2 -1699.535} C_VEL
LIN {X 0,Y 580.364,Z 817.77,A -85,B 0,C 180,E1 -1700.238,E2 -1700.238} C_VEL
LIN {X 0,Y 580.32,Z 826.013,A -85,B 0,C 180,E1 -1700.941,E2 -1700.941} C_VEL
LIN {X 0,Y 580.248,Z 834.542,A -85,B 0,C 180,E1 -1701.817,E2 -1701.817} C_VEL
LIN {X 0,Y 580.161,Z 841.622,A -85,B 0,C 180,E1 -1702.691,E2 -1702.691} C_VEL
LIN {X 0,Y 580.143,Z 848.569,A -85,B 0,C 180,E1 -1703.74,E2 -1703.74} C_VEL
LIN {X 0,Y 580.086,Z 854.133,A -85,B 0,C 180,E1 -1704.785,E2 -1704.785} C_VEL
LIN {X 0,Y 580.105,Z 858.498,A -85,B 0,C 180,E1 -1705.83,E2 -1705.83} C_VEL
LIN {X 0,Y 580.123,Z 860.819,A -85,B 0,C 180,E1 -1706.526,E2 -1706.526} C_VEL
LIN {X 0,Y 580.043,Z 862.692,A -85,B 0,C 180,E1 -1707.221,E2 -1707.221} C_VEL
LIN {X 0,Y 580.046,Z 865.132,A -85,B 0,C 180,E1 -1708.61,E2 -1708.61} C_VEL
LIN {X 0,Y 580.041,Z 865.753,A -85,B 0,C 180,E1 -1709.305,E2 -1709.305} C_VEL
LIN {X 0,Y 580.04,Z 865.815,A -85,B 0,C 180,E1 -1710.693,E2 -1710.693} C_VEL
LIN {X 0,Y 580.047,Z 865.236,A -85,B 0,C 180,E1 -1711.387,E2 -1711.387} C_VEL
LIN {X 0,Y 580.044,Z 862.917,A -85,B 0,C 180,E1 -1712.777,E2 -1712.777} C_VEL
LIN {X 0,Y 580.11,Z 860.043,A -85,B 0,C 180,E1 -1713.819,E2 -1713.819} C_VEL
LIN {X 0,Y 580.054,Z 856.145,A -85,B 0,C 180,E1 -1714.864,E2 -1714.864} C_VEL
LIN {X 0,Y 580.161,Z 851.116,A -85,B 0,C 180,E1 -1715.909,E2 -1715.909} C_VEL
LIN {X 0,Y 580.156,Z 844.781,A -85,B 0,C 180,E1 -1716.957,E2 -1716.957} C_VEL
LIN {X 0,Y 580.23,Z 836.85,A -85,B 0,C 180,E1 -1718.006,E2 -1718.006} C_VEL
LIN {X 0,Y 580.297,Z 828.78,A -85,B 0,C 180,E1 -1718.882,E2 -1718.882} C_VEL
LIN {X 0,Y 580.371,Z 819.995,A -85,B 0,C 180,E1 -1719.671,E2 -1719.671} C_VEL
LIN {X 0,Y 580.451,Z 810.536,A -85,B 0,C 180,E1 -1720.374,E2 -1720.374} C_VEL
LIN {X 0,Y 580.542,Z 800.388,A -85,B 0,C 180,E1 -1720.99,E2 -1720.99} C_VEL
LIN {X 0,Y 580.631,Z 789.171,A -85,B 0,C 180,E1 -1721.532,E2 -1721.532} C_VEL
LIN {X 0,Y 580.623,Z 781.563,A -85,B 0,C 180,E1 -1721.825,E2 -1721.825} C_VEL
LIN {X 0,Y 580.314,Z 780.198,A -85,B 0,C 180,E1 -1721.88,E2 -1721.88} C_VEL
LIN {X 0,Y 580.287,Z 780.196,A -85,B 0,C 180,E1 -1724.733,E2 -1724.733} C_VEL
LIN {X 0,Y 580.292,Z 780.206,A -85,B 0,C 180,E1 -1727.623,E2 -1727.623} C_VEL
LIN {X 0,Y 580.303,Z 780.203,A -85,B 0,C 180,E1 -1729.821,E2 -1729.821} C_VEL
LIN {X 0,Y 580.293,Z 780.195,A -85,B 0,C 180,E1 -1732.801,E2 -1732.801} C_VEL
LIN {X 0,Y 580.304,Z 780.194,A -85,B 0,C 180,E1 -1735.078,E2 -1735.078} C_VEL
LIN {X 0,Y 580.297,Z 780.201,A -85,B 0,C 180,E1 -1738.184,E2 -1738.184} C_VEL
LIN {X 0,Y 580.288,Z 780.196,A -85,B 0,C 180,E1 -1740.695,E2 -1740.695} C_VEL
LIN {X 0,Y 580.298,Z 780.195,A -85,B 0,C 180,E1 -1743.315,E2 -1743.315} C_VEL
LIN {X 0,Y 580.269,Z 780.202,A -85,B 0,C 180,E1 -1745.759,E2 -1745.759} C_VEL
LIN {X 0,Y 580.283,Z 780.207,A -85,B 0,C 180,E1 -1748.144,E2 -1748.144} C_VEL
LIN {X 0,Y 580.293,Z 780.196,A -85,B 0,C 180,E1 -1750.841,E2 -1750.841} C_VEL
LIN {X 0,Y 580.278,Z 780.198,A -85,B 0,C 180,E1 -1753.655,E2 -1753.655} C_VEL
LIN {X 0,Y 580.275,Z 780.203,A -85,B 0,C 180,E1 -1756.607,E2 -1756.607} C_VEL
LIN {X 0,Y 580.294,Z 780.196,A -85,B 0,C 180,E1 -1759.156,E2 -1759.156} C_VEL
LIN {X 0,Y 580.28,Z 780.197,A -85,B 0,C 180,E1 -1761.925,E2 -1761.925} C_VEL
LIN {X 0,Y 580.293,Z 780.203,A -85,B 0,C 180,E1 -1764.455,E2 -1764.455} C_VEL
LIN {X 0,Y 580.279,Z 780.202,A -85,B 0,C 180,E1 -1766.974,E2 -1766.974} C_VEL
LIN {X 0,Y 580.296,Z 780.195,A -85,B 0,C 180,E1 -1769.425,E2 -1769.425} C_VEL
LIN {X 0,Y 580.283,Z 780.197,A -85,B 0,C 180,E1 -1772.14,E2 -1772.14} C_VEL
LIN {X 0,Y 580.296,Z 780.204,A -85,B 0,C 180,E1 -1774.92,E2 -1774.92} C_VEL
LIN {X 0,Y 580.257,Z 780.199,A -85,B 0,C 180,E1 -1777.947,E2 -1777.947} C_VEL
LIN {X 0,Y 580.302,Z 780.203,A -85,B 0,C 180,E1 -1780.913,E2 -1780.913} C_VEL
LIN {X 0,Y 580.26,Z 780.199,A -85,B 0,C 180,E1 -1783.825,E2 -1783.825} C_VEL
LIN {X 0,Y 580.309,Z 780.193,A -85,B 0,C 180,E1 -1785.983,E2 -1785.983} C_VEL
LIN {X 0,Y 580.373,Z 780.189,A -85,B 0,C 180,E1 -1788.828,E2 -1788.828} C_VEL
LIN {X 0,Y 580.315,Z 780.196,A -85,B 0,C 180,E1 -1791.644,E2 -1791.644} C_VEL
LIN {X 0,Y 580.308,Z 780.193,A -85,B 0,C 180,E1 -1794.44,E2 -1794.44} C_VEL
LIN {X 0,Y 580.337,Z 780.196,A -85,B 0,C 180,E1 -1797.223,E2 -1797.223} C_VEL
LIN {X 0,Y 580.321,Z 780.194,A -85,B 0,C 180,E1 -1800,E2 -1800} C_VEL
LIN {X 0,Y 580.317,Z 780.193,A -85,B 0,C 180,E1 -1802.777,E2 -1802.777} C_VEL
LIN {X 0,Y 580.312,Z 780.203,A -85,B 0,C 180,E1 -1805.56,E2 -1805.56} C_VEL
LIN {X 0,Y 580.307,Z 780.194,A -85,B 0,C 180,E1 -1808.356,E2 -1808.356} C_VEL
LIN {X 0,Y 580.281,Z 780.198,A -85,B 0,C 180,E1 -1811.191,E2 -1811.191} C_VEL
LIN {X 0,Y 580.298,Z 780.202,A -85,B 0,C 180,E1 -1814.018,E2 -1814.018} C_VEL
LIN {X 0,Y 580.271,Z 780.198,A -85,B 0,C 180,E1 -1816.907,E2 -1816.907} C_VEL
LIN {X 0,Y 580.265,Z 780.207,A -85,B 0,C 180,E1 -1819.824,E2 -1819.824} C_VEL
LIN {X 0,Y 580.249,Z 780.211,A -85,B 0,C 180,E1 -1822.054,E2 -1822.054} C_VEL
LIN {X 0,Y 580.284,Z 780.196,A -85,B 0,C 180,E1 -1825.081,E2 -1825.081} C_VEL
LIN {X 0,Y 580.26,Z 780.21,A -85,B 0,C 180,E1 -1828.188,E2 -1828.188} C_VEL
LIN {X 0,Y 580.27,Z 780.201,A -85,B 0,C 180,E1 -1830.696,E2 -1830.696} C_VEL
LIN {X 0,Y 580.265,Z 780.198,A -85,B 0,C 180,E1 -1833.314,E2 -1833.314} C_VEL
LIN {X 0,Y 580.211,Z 780.207,A -85,B 0,C 180,E1 -1835.755,E2 -1835.755} C_VEL
LIN {X 0,Y 580.262,Z 780.205,A -85,B 0,C 180,E1 -1838.149,E2 -1838.149} C_VEL
LIN {X 0,Y 580.26,Z 780.204,A -85,B 0,C 180,E1 -1840.847,E2 -1840.847} C_VEL
LIN {X 0,Y 580.228,Z 780.204,A -85,B 0,C 180,E1 -1843.388,E2 -1843.388} C_VEL
LIN {X 0,Y 580.214,Z 780.211,A -85,B 0,C 180,E1 -1846.339,E2 -1846.339} C_VEL
LIN {X 0,Y 580.244,Z 780.205,A -85,B 0,C 180,E1 -1849.154,E2 -1849.154} C_VEL
LIN {X 0,Y 580.26,Z 780.202,A -85,B 0,C 180,E1 -1851.931,E2 -1851.931} C_VEL
LIN {X 0,Y 580.275,Z 780.302,A -85,B 0,C 180,E1 -1853.177,E2 -1853.177} C_VEL
LIN {X 0,Y 581.115,Z 784.758,A -85,B 0,C 180,E1 -1854.125,E2 -1854.125} C_VEL
LIN {X 0,Y 581.302,Z 796.877,A -85,B 0,C 180,E1 -1856.535,E2 -1856.535} C_VEL
LIN {X 0,Y 581.134,Z 811.157,A -85,B 0,C 180,E1 -1859.476,E2 -1859.476} C_VEL
LIN {X 0,Y 580.905,Z 825.296,A -85,B 0,C 180,E1 -1862.329,E2 -1862.329} C_VEL
LIN {X 0,Y 580.778,Z 839.719,A -85,B 0,C 180,E1 -1865.173,E2 -1865.173} C_VEL
LIN {X 0,Y 580.639,Z 852.242,A -85,B 0,C 180,E1 -1867.589,E2 -1867.589} C_VEL
LIN {X 0,Y 580.489,Z 867.822,A -85,B 0,C 180,E1 -1870.541,E2 -1870.541} C_VEL
LIN {X 0,Y 580.416,Z 881.587,A -85,B 0,C 180,E1 -1873.107,E2 -1873.107} C_VEL
LIN {X 0,Y 580.249,Z 897.238,A -85,B 0,C 180,E1 -1875.983,E2 -1875.983} C_VEL
LIN {X 0,Y 580.265,Z 906.189,A -85,B 0,C 180,E1 -1877.609,E2 -1877.609} C_VEL
LIN {X 0,Y 580.82,Z 912.021,A -85,B 0,C 180,E1 -1877.71,E2 -1877.71} C_VEL
LIN {X 0,Y 580.721,Z 925.264,A -85,B 0,C 180,E1 -1878.018,E2 -1878.018} C_VEL
LIN {X 0,Y 580.629,Z 938.525,A -85,B 0,C 180,E1 -1878.481,E2 -1878.481} C_VEL
LIN {X 0,Y 580.583,Z 949.658,A -85,B 0,C 180,E1 -1879.01,E2 -1879.01} C_VEL
LIN {X 0,Y 580.421,Z 961.221,A -85,B 0,C 180,E1 -1879.713,E2 -1879.713} C_VEL
LIN {X 0,Y 580.346,Z 971.613,A -85,B 0,C 180,E1 -1880.504,E2 -1880.504} C_VEL
LIN {X 0,Y 580.262,Z 980.045,A -85,B 0,C 180,E1 -1881.293,E2 -1881.293} C_VEL
LIN {X 0,Y 580.221,Z 987.972,A -85,B 0,C 180,E1 -1882.169,E2 -1882.169} C_VEL
LIN {X 0,Y 580.155,Z 995.642,A -85,B 0,C 180,E1 -1883.22,E2 -1883.22} C_VEL
LIN {X 0,Y 580.139,Z 1002.687,A -85,B 0,C 180,E1 -1884.44,E2 -1884.44} C_VEL
LIN {X 0,Y 580.108,Z 1007.376,A -85,B 0,C 180,E1 -1885.485,E2 -1885.485} C_VEL
LIN {X 0,Y 580.122,Z 1010.961,A -85,B 0,C 180,E1 -1886.529,E2 -1886.529} C_VEL
LIN {X 0,Y 580.043,Z 1012.813,A -85,B 0,C 180,E1 -1887.223,E2 -1887.223} C_VEL
LIN {X 0,Y 580.038,Z 1014.203,A -85,B 0,C 180,E1 -1887.918,E2 -1887.918} C_VEL
LIN {X 0,Y 580.04,Z 1015.785,A -85,B 0,C 180,E1 -1889.307,E2 -1889.307} C_VEL
LIN {X 0,Y 580.037,Z 1016,A -85,B 0,C 180,E1 -1890.001,E2 -1890.001} C_VEL
LIN {X 0,Y 580.046,Z 1015.183,A -85,B 0,C 180,E1 -1891.39,E2 -1891.39} C_VEL
LIN {X 0,Y 580.038,Z 1014.199,A -85,B 0,C 180,E1 -1892.084,E2 -1892.084} C_VEL
LIN {X 0,Y 580.043,Z 1012.806,A -85,B 0,C 180,E1 -1892.779,E2 -1892.779} C_VEL
LIN {X 0,Y 580.109,Z 1009.892,A -85,B 0,C 180,E1 -1893.822,E2 -1893.822} C_VEL
LIN {X 0,Y 580.053,Z 1005.945,A -85,B 0,C 180,E1 -1894.866,E2 -1894.866} C_VEL
LIN {X 0,Y 580.14,Z 999.871,A -85,B 0,C 180,E1 -1896.086,E2 -1896.086} C_VEL
LIN {X 0,Y 580.185,Z 993.228,A -85,B 0,C 180,E1 -1897.134,E2 -1897.134} C_VEL
LIN {X 0,Y 580.247,Z 984.98,A -85,B 0,C 180,E1 -1898.183,E2 -1898.183} C_VEL
LIN {X 0,Y 580.334,Z 974.588,A -85,B 0,C 180,E1 -1899.235,E2 -1899.235} C_VEL
LIN {X 0,Y 580.433,Z 964.915,A -85,B 0,C 180,E1 -1900.025,E2 -1900.025} C_VEL
LIN {X 0,Y 580.543,Z 954.308,A -85,B 0,C 180,E1 -1900.728,E2 -1900.728} C_VEL
LIN {X 0,Y 580.626,Z 941.773,A -85,B 0,C 180,E1 -1901.375,E2 -1901.375} C_VEL
LIN {X 0,Y 580.721,Z 928.846,A -85,B 0,C 180,E1 -1901.874,E2 -1901.874} C_VEL
LIN {X 0,Y 580.796,Z 916.456,A -85,B 0,C 180,E1 -1902.204,E2 -1902.204} C_VEL
LIN {X 0,Y 580.539,Z 908.093,A -85,B 0,C 180,E1 -1902.357,E2 -1902.357} C_VEL
LIN {X 0,Y 580.25,Z 906.028,A -85,B 0,C 180,E1 -1902.416,E2 -1902.416} C_VEL
LIN {X 0,Y 580.316,Z 889.399,A -85,B 0,C 180,E1 -1905.453,E2 -1905.453} C_VEL
LIN {X 0,Y 580.435,Z 875.704,A -85,B 0,C 180,E1 -1907.985,E2 -1907.985} C_VEL
LIN {X 0,Y 580.542,Z 862.01,A -85,B 0,C 180,E1 -1910.554,E2 -1910.554} C_VEL
LIN {X 0,Y 580.691,Z 847.761,A -85,B 0,C 180,E1 -1913.27,E2 -1913.27} C_VEL
LIN {X 0,Y 580.85,Z 834.62,A -85,B 0,C 180,E1 -1915.823,E2 -1915.823} C_VEL
LIN {X 0,Y 580.999,Z 818.969,A -85,B 0,C 180,E1 -1918.938,E2 -1918.938} C_VEL
LIN {X 0,Y 581.185,Z 807.231,A -85,B 0,C 180,E1 -1921.332,E2 -1921.332} C_VEL
LIN {X 0,Y 581.298,Z 795.186,A -85,B 0,C 180,E1 -1923.791,E2 -1923.791} C_VEL
LIN {X 0,Y 581.132,Z 784.697,A -85,B 0,C 180,E1 -1925.877,E2 -1925.877} C_VEL
LIN {X 0,Y 580.272,Z 780.208,A -85,B 0,C 180,E1 -1926.867,E2 -1926.867} C_VEL
LIN {X 0,Y 580.252,Z 780.203,A -85,B 0,C 180,E1 -1929.937,E2 -1929.937} C_VEL
LIN {X 0,Y 580.213,Z 780.207,A -85,B 0,C 180,E1 -1932.713,E2 -1932.713} C_VEL
LIN {X 0,Y 580.22,Z 780.214,A -85,B 0,C 180,E1 -1935.369,E2 -1935.369} C_VEL
LIN {X 0,Y 580.227,Z 780.205,A -85,B 0,C 180,E1 -1938.226,E2 -1938.226} C_VEL
LIN {X 0,Y 580.232,Z 780.203,A -85,B 0,C 180,E1 -1940.961,E2 -1940.961} C_VEL
LIN {X 0,Y 580.208,Z 780.214,A -85,B 0,C 180,E1 -1943.592,E2 -1943.592} C_VEL
LIN {X 0,Y 580.261,Z 780.204,A -85,B 0,C 180,E1 -1946.142,E2 -1946.142} C_VEL
LIN {X 0,Y 580.236,Z 780.203,A -85,B 0,C 180,E1 -1948.612,E2 -1948.612} C_VEL
LIN {X 0,Y 580.24,Z 780.202,A -85,B 0,C 180,E1 -1951.021,E2 -1951.021} C_VEL
LIN {X 0,Y 580.24,Z 780.212,A -85,B 0,C 180,E1 -1954.148,E2 -1954.148} C_VEL
LIN {X 0,Y 580.226,Z 780.203,A -85,B 0,C 180,E1 -1957.008,E2 -1957.008} C_VEL
LIN {X 0,Y 580.233,Z 780.203,A -85,B 0,C 180,E1 -1959.436,E2 -1959.436} C_VEL
LIN {X 0,Y 580.228,Z 780.214,A -85,B 0,C 180,E1 -1962.373,E2 -1962.373} C_VEL
LIN {X 0,Y 580.253,Z 780.201,A -85,B 0,C 180,E1 -1965.265,E2 -1965.265} C_VEL
LIN {X 0,Y 580.271,Z 780.204,A -85,B 0,C 180,E1 -1968.207,E2 -1968.207} C_VEL
LIN {X 0,Y 580.66,Z 783.903,A -85,B 0,C 180,E1 -1968.348,E2 -1968.348} C_VEL
LIN {X 0,Y 580.478,Z 796.604,A -85,B 0,C 180,E1 -1968.896,E2 -1968.896} C_VEL
LIN {X 0,Y 580.417,Z 807.875,A -85,B 0,C 180,E1 -1969.535,E2 -1969.535} C_VEL
LIN {X 0,Y 580.36,Z 817.796,A -85,B 0,C 180,E1 -1970.239,E2 -1970.239} C_VEL
LIN {X 0,Y 580.306,Z 826.025,A -85,B 0,C 180,E1 -1970.942,E2 -1970.942} C_VEL
LIN {X 0,Y 580.242,Z 836.093,A -85,B 0,C 180,E1 -1971.993,E2 -1971.993} C_VEL
LIN {X 0,Y 580.159,Z 844.154,A -85,B 0,C 180,E1 -1973.042,E2 -1973.042} C_VEL
LIN {X 0,Y 580.165,Z 850.617,A -85,B 0,C 180,E1 -1974.09,E2 -1974.09} C_VEL
LIN {X 0,Y 580.053,Z 855.746,A -85,B 0,C 180,E1 -1975.135,E2 -1975.135} C_VEL
LIN {X 0,Y 580.109,Z 859.732,A -85,B 0,C 180,E1 -1976.179,E2 -1976.179} C_VEL
LIN {X 0,Y 580.043,Z 862.688,A -85,B 0,C 180,E1 -1977.222,E2 -1977.222} C_VEL
LIN {X 0,Y 580.038,Z 864.133,A -85,B 0,C 180,E1 -1977.917,E2 -1977.917} C_VEL
LIN {X 0,Y 580.041,Z 865.755,A -85,B 0,C 180,E1 -1979.306,E2 -1979.306} C_VEL
LIN {X 0,Y 580.038,Z 865.996,A -85,B 0,C 180,E1 -1980,E2 -1980} C_VEL
LIN {X 0,Y 580.047,Z 865.231,A -85,B 0,C 180,E1 -1981.389,E2 -1981.389} C_VEL
LIN {X 0,Y 580.037,Z 864.276,A -85,B 0,C 180,E1 -1982.083,E2 -1982.083} C_VEL
LIN {X 0,Y 580.044,Z 862.884,A -85,B 0,C 180,E1 -1982.778,E2 -1982.778} C_VEL
LIN {X 0,Y 580.11,Z 860.01,A -85,B 0,C 180,E1 -1983.821,E2 -1983.821} C_VEL
LIN {X 0,Y 580.053,Z 856.113,A -85,B 0,C 180,E1 -1984.865,E2 -1984.865} C_VEL
LIN {X 0,Y 580.16,Z 851.089,A -85,B 0,C 180,E1 -1985.91,E2 -1985.91} C_VEL
LIN {X 0,Y 580.158,Z 844.778,A -85,B 0,C 180,E1 -1986.958,E2 -1986.958} C_VEL
LIN {X 0,Y 580.242,Z 836.858,A -85,B 0,C 180,E1 -1988.007,E2 -1988.007} C_VEL
LIN {X 0,Y 580.306,Z 826.962,A -85,B 0,C 180,E1 -1989.058,E2 -1989.058} C_VEL
LIN {X 0,Y 580.382,Z 816.692,A -85,B 0,C 180,E1 -1989.937,E2 -1989.937} C_VEL
LIN {X 0,Y 580.451,Z 805.112,A -85,B 0,C 180,E1 -1990.726,E2 -1990.726} C_VEL
LIN {X 0,Y 580.549,Z 794.147,A -85,B 0,C 180,E1 -1991.312,E2 -1991.312} C_VEL
LIN {X 0,Y 580.634,Z 782.937,A -85,B 0,C 180,E1 -1991.777,E2 -1991.777} C_VEL
LIN {X 0,Y 580.3,Z 780.2,A -85,B 0,C 180,E1 -1991.881,E2 -1991.881} C_VEL
LIN {X 0,Y 580.256,Z 780.201,A -85,B 0,C 180,E1 -1994.735,E2 -1994.735} C_VEL
LIN {X 0,Y 580.219,Z 780.212,A -85,B 0,C 180,E1 -1997.464,E2 -1997.464} C_VEL
LIN {X 0,Y 579.569,Z 780.299,A -85,B 0,C 180,E1 -1998.044,E2 -1998.044} C_VEL
LIN {X 0,Y 576.705,Z 780.654,A -85,B 0,C 180,E1 -1998.984,E2 -1998.984} C_VEL
LIN {X 0,Y 574.283,Z 780.952,A -85,B 0,C 180,E1 -1999.741,E2 -1999.741} C_VEL
LIN {X 0,Y 573.257,Z 781.072,A -85,B 0,C 180,E1 -2000.325,E2 -2000.325} C_VEL
LIN {X 0,Y 573.182,Z 781.08,A -85,B 0,C 180,E1 -2000.523,E2 -2000.523} C_VEL
LIN {X 0,Y 573.182,Z 781.082,A -85,B 0,C 180,E1 -2003.131,E2 -2003.131} C_VEL
LIN {X 0,Y 573.209,Z 781.082,A -85,B 0,C 180,E1 -2005.412,E2 -2005.412} C_VEL
LIN {X 0,Y 573.19,Z 781.085,A -85,B 0,C 180,E1 -2008.016,E2 -2008.016} C_VEL
LIN {X 0,Y 573.221,Z 781.075,A -85,B 0,C 180,E1 -2010.88,E2 -2010.88} C_VEL
LIN {X 0,Y 573.247,Z 781.076,A -85,B 0,C 180,E1 -2013.52,E2 -2013.52} C_VEL
LIN {X 0,Y 573.187,Z 781.087,A -85,B 0,C 180,E1 -2016.054,E2 -2016.054} C_VEL
LIN {X 0,Y 573.234,Z 781.074,A -85,B 0,C 180,E1 -2018.702,E2 -2018.702} C_VEL
LIN {X 0,Y 573.207,Z 781.08,A -85,B 0,C 180,E1 -2021.459,E2 -2021.459} C_VEL
LIN {X 0,Y 573.222,Z 781.081,A -85,B 0,C 180,E1 -2024.335,E2 -2024.335} C_VEL
LIN {X 0,Y 573.213,Z 781.079,A -85,B 0,C 180,E1 -2026.638,E2 -2026.638} C_VEL
LIN {X 0,Y 573.251,Z 781.073,A -85,B 0,C 180,E1 -2029.475,E2 -2029.475} C_VEL
LIN {X 0,Y 573.234,Z 781.084,A -85,B 0,C 180,E1 -2032.191,E2 -2032.191} C_VEL
LIN {X 0,Y 573.235,Z 781.074,A -85,B 0,C 180,E1 -2035.229,E2 -2035.229} C_VEL
LIN {X 0,Y 573.242,Z 781.083,A -85,B 0,C 180,E1 -2038.184,E2 -2038.184} C_VEL
LIN {X 0,Y 573.248,Z 781.077,A -85,B 0,C 180,E1 -2040.632,E2 -2040.632} C_VEL
LIN {X 0,Y 573.223,Z 781.076,A -85,B 0,C 180,E1 -2043.022,E2 -2043.022} C_VEL
LIN {X 0,Y 573.241,Z 781.072,A -85,B 0,C 180,E1 -2045.364,E2 -2045.364} C_VEL
LIN {X 0,Y 573.239,Z 781.074,A -85,B 0,C 180,E1 -2047.661,E2 -2047.661} C_VEL
LIN {X 0,Y 573.273,Z 781.078,A -85,B 0,C 180,E1 -2050.669,E2 -2050.669} C_VEL
LIN {X 0,Y 573.251,Z 781.073,A -85,B 0,C 180,E1 -2053.621,E2 -2053.621} C_VEL
LIN {X 0,Y 573.271,Z 781.071,A -85,B 0,C 180,E1 -2055.806,E2 -2055.806} C_VEL
LIN {X 0,Y 573.276,Z 781.074,A -85,B 0,C 180,E1 -2058.082,E2 -2058.082} C_VEL
LIN {X 0,Y 573.719,Z 785.132,A -85,B 0,C 180,E1 -2058.248,E2 -2058.248} C_VEL
LIN {X 0,Y 573.588,Z 797.834,A -85,B 0,C 180,E1 -2058.824,E2 -2058.824} C_VEL
LIN {X 0,Y 573.465,Z 809.156,A -85,B 0,C 180,E1 -2059.495,E2 -2059.495} C_VEL
LIN {X 0,Y 573.355,Z 818.847,A -85,B 0,C 180,E1 -2060.207,E2 -2060.207} C_VEL
LIN {X 0,Y 573.262,Z 827.818,A -85,B 0,C 180,E1 -2061.006,E2 -2061.006} C_VEL
LIN {X 0,Y 573.177,Z 836.052,A -85,B 0,C 180,E1 -2061.893,E2 -2061.893} C_VEL
LIN {X 0,Y 573.115,Z 842.878,A -85,B 0,C 180,E1 -2062.778,E2 -2062.778} C_VEL
LIN {X 0,Y 573.068,Z 849.597,A -85,B 0,C 180,E1 -2063.839,E2 -2063.839} C_VEL
LIN {X 0,Y 573.009,Z 854.125,A -85,B 0,C 180,E1 -2064.721,E2 -2064.721} C_VEL
LIN {X 0,Y 573.031,Z 858.49,A -85,B 0,C 180,E1 -2065.779,E2 -2065.779} C_VEL
LIN {X 0,Y 573.022,Z 860.819,A -85,B 0,C 180,E1 -2066.483,E2 -2066.483} C_VEL
LIN {X 0,Y 572.959,Z 862.693,A -85,B 0,C 180,E1 -2067.186,E2 -2067.186} C_VEL
LIN {X 0,Y 572.945,Z 865.132,A -85,B 0,C 180,E1 -2068.593,E2 -2068.593} C_VEL
LIN {X 0,Y 572.941,Z 865.754,A -85,B 0,C 180,E1 -2069.296,E2 -2069.296} C_VEL
LIN {X 0,Y 572.94,Z 865.815,A -85,B 0,C 180,E1 -2070.702,E2 -2070.702} C_VEL
LIN {X 0,Y 572.946,Z 865.234,A -85,B 0,C 180,E1 -2071.404,E2 -2071.404} C_VEL
LIN {X 0,Y 572.959,Z 862.916,A -85,B 0,C 180,E1 -2072.811,E2 -2072.811} C_VEL
LIN {X 0,Y 573.014,Z 860.042,A -85,B 0,C 180,E1 -2073.867,E2 -2073.867} C_VEL
LIN {X 0,Y 572.963,Z 856.144,A -85,B 0,C 180,E1 -2074.924,E2 -2074.924} C_VEL
LIN {X 0,Y 573.07,Z 850.126,A -85,B 0,C 180,E1 -2076.159,E2 -2076.159} C_VEL
LIN {X 0,Y 573.112,Z 843.536,A -85,B 0,C 180,E1 -2077.219,E2 -2077.219} C_VEL
LIN {X 0,Y 573.168,Z 836.84,A -85,B 0,C 180,E1 -2078.105,E2 -2078.105} C_VEL
LIN {X 0,Y 573.25,Z 828.761,A -85,B 0,C 180,E1 -2078.992,E2 -2078.992} C_VEL
LIN {X 0,Y 573.354,Z 819.973,A -85,B 0,C 180,E1 -2079.791,E2 -2079.791} C_VEL
LIN {X 0,Y 573.463,Z 810.511,A -85,B 0,C 180,E1 -2080.502,E2 -2080.502} C_VEL
LIN {X 0,Y 573.556,Z 800.518,A -85,B 0,C 180,E1 -2081.117,E2 -2081.117} C_VEL
LIN {X 0,Y 573.654,Z 790.67,A -85,B 0,C 180,E1 -2081.606,E2 -2081.606} C_VEL
LIN {X 0,Y 573.617,Z 782.695,A -85,B 0,C 180,E1 -2081.931,E2 -2081.931} C_VEL
LIN {X 0,Y 573.26,Z 781.076,A -85,B 0,C 180,E1 -2082.006,E2 -2082.006} C_VEL
LIN {X 0,Y 573.235,Z 781.076,A -85,B 0,C 180,E1 -2084.918,E2 -2084.918} C_VEL
LIN {X 0,Y 573.243,Z 781.081,A -85,B 0,C 180,E1 -2087.847,E2 -2087.847} C_VEL
LIN {X 0,Y 573.25,Z 781.077,A -85,B 0,C 180,E1 -2090.075,E2 -2090.075} C_VEL
LIN {X 0,Y 573.232,Z 781.075,A -85,B 0,C 180,E1 -2093.098,E2 -2093.098} C_VEL
LIN {X 0,Y 573.252,Z 781.075,A -85,B 0,C 180,E1 -2095.408,E2 -2095.408} C_VEL
LIN {X 0,Y 573.26,Z 781.08,A -85,B 0,C 180,E1 -2098.03,E2 -2098.03} C_VEL
LIN {X 0,Y 573.234,Z 781.074,A -85,B 0,C 180,E1 -2100.882,E2 -2100.882} C_VEL
LIN {X 0,Y 573.256,Z 781.074,A -85,B 0,C 180,E1 -2103.522,E2 -2103.522} C_VEL
LIN {X 0,Y 573.238,Z 781.083,A -85,B 0,C 180,E1 -2106.048,E2 -2106.048} C_VEL
LIN {X 0,Y 573.241,Z 781.076,A -85,B 0,C 180,E1 -2108.699,E2 -2108.699} C_VEL
LIN {X 0,Y 573.245,Z 781.074,A -85,B 0,C 180,E1 -2111.594,E2 -2111.594} C_VEL
LIN {X 0,Y 573.229,Z 781.086,A -85,B 0,C 180,E1 -2114.331,E2 -2114.331} C_VEL
LIN {X 0,Y 573.233,Z 781.073,A -85,B 0,C 180,E1 -2117.357,E2 -2117.357} C_VEL
LIN {X 0,Y 573.238,Z 781.083,A -85,B 0,C 180,E1 -2120.392,E2 -2120.392} C_VEL
LIN {X 0,Y 573.244,Z 781.075,A -85,B 0,C 180,E1 -2123.077,E2 -2123.077} C_VEL
